    REGION Cartesian_Jog
        // HMI jog buttons -> GDB_AxisCtrl.LKinCtrl.input.jogframe Cartesian
        // direction bits. WCS frame jog: the 4 HMI axis-pairs drive
        // X (J1 buttons) / Y (J2) / Z (J3) / A (J4). XOR safety - if both
        // forward + backward are held, neither wins. Each bit is ANDed with
        // statManualOK, so leaving manual mode forces every jog bit FALSE.
        // SCARA is 4-DOF: the B / C jog directions are held FALSE.
        "GDB_AxisCtrl".LKinCtrl.input.jogframe."jogX+" := #statManualOK AND "GDB_ManualCmd".bo_J1_JogForward  AND NOT "GDB_ManualCmd".bo_J1_JogBackward;
        "GDB_AxisCtrl".LKinCtrl.input.jogframe."jogX-" := #statManualOK AND "GDB_ManualCmd".bo_J1_JogBackward AND NOT "GDB_ManualCmd".bo_J1_JogForward;
        "GDB_AxisCtrl".LKinCtrl.input.jogframe."jogY+" := #statManualOK AND "GDB_ManualCmd".bo_J2_JogForward  AND NOT "GDB_ManualCmd".bo_J2_JogBackward;
        "GDB_AxisCtrl".LKinCtrl.input.jogframe."jogY-" := #statManualOK AND "GDB_ManualCmd".bo_J2_JogBackward AND NOT "GDB_ManualCmd".bo_J2_JogForward;
        "GDB_AxisCtrl".LKinCtrl.input.jogframe."jogZ+" := #statManualOK AND "GDB_ManualCmd".bo_J3_JogForward  AND NOT "GDB_ManualCmd".bo_J3_JogBackward;
        "GDB_AxisCtrl".LKinCtrl.input.jogframe."jogZ-" := #statManualOK AND "GDB_ManualCmd".bo_J3_JogBackward AND NOT "GDB_ManualCmd".bo_J3_JogForward;
        "GDB_AxisCtrl".LKinCtrl.input.jogframe."jogA+" := #statManualOK AND "GDB_ManualCmd".bo_J4_JogForward  AND NOT "GDB_ManualCmd".bo_J4_JogBackward;
        "GDB_AxisCtrl".LKinCtrl.input.jogframe."jogA-" := #statManualOK AND "GDB_ManualCmd".bo_J4_JogBackward AND NOT "GDB_ManualCmd".bo_J4_JogForward;
        "GDB_AxisCtrl".LKinCtrl.input.jogframe."jogB+" := FALSE;
        "GDB_AxisCtrl".LKinCtrl.input.jogframe."jogB-" := FALSE;
        "GDB_AxisCtrl".LKinCtrl.input.jogframe."jogC+" := FALSE;
        "GDB_AxisCtrl".LKinCtrl.input.jogframe."jogC-" := FALSE;
    END_REGION

    REGION Kin_Manual_Move
        // bo_KinGo rising edge -> a point-to-point move to the operator-set
        // (cfgKinTargetX/Y/Z/A) via the shared movelinear interface (the
        // OB30 axis layer runs the MC). The R_TRIG runs every scan; the move
        // is issued only in manual mode. bo_execute is held until FB_AxisCtrl
        // reports the move done. Manual dynamics: 200 mm/s (auto cycle: 300).
        #sRTRIGKinGo(CLK := "GDB_ManualCmd".bo_KinGo);
        IF #statManualOK THEN
            IF #sRTRIGKinGo.Q THEN
                "GDB_AxisCtrl".LKinCtrl.input.movelinear.targetposition.x := "GDB_ManualCmd".cfgKinTargetX;
                "GDB_AxisCtrl".LKinCtrl.input.movelinear.targetposition.y := "GDB_ManualCmd".cfgKinTargetY;
                "GDB_AxisCtrl".LKinCtrl.input.movelinear.targetposition.z := "GDB_ManualCmd".cfgKinTargetZ;
                "GDB_AxisCtrl".LKinCtrl.input.movelinear.targetposition.a := "GDB_ManualCmd".cfgKinTargetA;
                "GDB_AxisCtrl".LKinCtrl.input.movelinear.targetposition.b := 0.0;
                "GDB_AxisCtrl".LKinCtrl.input.movelinear.targetposition.c := 0.0;
                "GDB_AxisCtrl".LKinCtrl.input.movelinear.r64_velocity     := 200.0;
                "GDB_AxisCtrl".LKinCtrl.input.movelinear.r64_acceleration := 2000.0;
                "GDB_AxisCtrl".LKinCtrl.input.movelinear.r64_deceleration := 2000.0;
                "GDB_AxisCtrl".LKinCtrl.input.movelinear.r64_jerk         := 20000.0;
                "GDB_AxisCtrl".LKinCtrl.input.movelinear.bo_isPTP         := FALSE;
                "GDB_AxisCtrl".LKinCtrl.input.movelinear.bo_execute       := TRUE;
            END_IF;
            // drop the execute hold once the OB30 axis layer reports done
            IF "GDB_AxisCtrl".LKinCtrl.output.movelinear.bo_done THEN
                "GDB_AxisCtrl".LKinCtrl.input.movelinear.bo_execute := FALSE;
            END_IF;
        END_IF;
    END_REGION

    REGION Status_Mirror
        // TO StatusWord bits + GDB_AxisCtrl outputs -> GDB_ManualStatus.
        // Runs every scan (NOT gated on statManualOK) so HMI lamps show the
        // truth regardless of mode. StatusWord (Siemens TO_PositioningAxis
        // MC 9.0): %X1 = Error, %X5 = Homed, %X7 = Standstill (NOT-%X7 =
        // motion in progress). Group power is all-or-nothing
        // (LKinCtrl_MC_GroupPower) - all 4 joints mirror the group bo_enabled.
        "GDB_ManualStatus".bo_J1_Enabled := "GDB_AxisCtrl".LKinCtrl.output.bo_enabled;
        "GDB_ManualStatus".bo_J2_Enabled := "GDB_AxisCtrl".LKinCtrl.output.bo_enabled;
        "GDB_ManualStatus".bo_J3_Enabled := "GDB_AxisCtrl".LKinCtrl.output.bo_enabled;
        "GDB_ManualStatus".bo_J4_Enabled := "GDB_AxisCtrl".LKinCtrl.output.bo_enabled;

        "GDB_ManualStatus".bo_J1_Homed := "J1_SCARA_Arm3D".StatusWord.%X5;
        "GDB_ManualStatus".bo_J2_Homed := "J2_SCARA_Arm3D".StatusWord.%X5;
        "GDB_ManualStatus".bo_J3_Homed := "J3_SCARA_Arm3D".StatusWord.%X5;
        "GDB_ManualStatus".bo_J4_Homed := "J4_SCARA_Arm3D".StatusWord.%X5;

        "GDB_ManualStatus".bo_J1_Error := "J1_SCARA_Arm3D".StatusWord.%X1;
        "GDB_ManualStatus".bo_J2_Error := "J2_SCARA_Arm3D".StatusWord.%X1;
        "GDB_ManualStatus".bo_J3_Error := "J3_SCARA_Arm3D".StatusWord.%X1;
        "GDB_ManualStatus".bo_J4_Error := "J4_SCARA_Arm3D".StatusWord.%X1;

        "GDB_ManualStatus".bo_J1_JogActive := NOT "J1_SCARA_Arm3D".StatusWord.%X7;
        "GDB_ManualStatus".bo_J2_JogActive := NOT "J2_SCARA_Arm3D".StatusWord.%X7;
        "GDB_ManualStatus".bo_J3_JogActive := NOT "J3_SCARA_Arm3D".StatusWord.%X7;
        "GDB_ManualStatus".bo_J4_JogActive := NOT "J4_SCARA_Arm3D".StatusWord.%X7;

        "GDB_ManualStatus".bo_KinEnabled := "GDB_AxisCtrl".LKinCtrl.output.bo_enabled;
        "GDB_ManualStatus".bo_KinHomed   := "GDB_AxisCtrl".LKinCtrl.output.bo_homed;
        "GDB_ManualStatus".bo_KinError   := "GDB_AxisCtrl".LKinCtrl.output.bo_fault;
        "GDB_ManualStatus".bo_KinReady   := "GDB_AxisCtrl".LKinCtrl.output.bo_ready;
        "GDB_ManualStatus".bo_KinManualBusy := "GDB_AxisCtrl".LKinCtrl.output.movelinear.bo_busy;
    END_REGION

END_FUNCTION_BLOCK

FUNCTION_BLOCK "FB_Init"
{ S7_Optimized_Access := 'TRUE' }
VERSION : 1.0
// =====================================================================
// SCARA ABCDE — Initialization / Homing  (Phase 3, 2026-05-21)
//
// Dedicated init/homing block per the 2026-05-21 TIA programming review
// (§1.4): homing must NOT live inside FB_AutoCtrl. Belongs to the 600
// axis/kinematics layer and runs in OB30 (10 ms cyclic interrupt),
// alongside FB_AxisCtrl.
//
// Homes the SCARA kinematics group via the library FB
// LKinCtrl_MC_GroupHome, which fires MC_HOME on every axis of ScaraArm3D
// from a per-axis mode[] + position[] array — read straight from the
// consolidated GDB_AxisCtrl.LKinCtrl.input.configuration.home struct.
//
// Two home types (review item E) — selected by the i16_mode[] value
// (the HMI / Startup OB sets it; FB_Init is mode-agnostic):
//   mode = 5  "go to zero position" — MC_Home active homing: each axis
//             runs its configured homing movement and ends at the TO
//             <TO>.Homing.HomePosition.
//   mode = 7  "set current as home" — MC_Home absolute-encoder
//             adjustment (absolute): current position set to
//             position[i], offset stored retentively. Correct for the
//             SCARA's absolute encoders (Sensor[1].Type = 2); no motion.
//
// Trigger: rising edge of GDB_AxisCtrl.LKinCtrl.input.bo_home (the HMI
// Home button). LKinCtrl_MC_GroupHome edge-detects 'execute' internally.
//
// TODO (Phase 3 refinement): for mode = 5 active homing, sequence the
// per-axis homing order + speeds (the review asks for an explicit axis
// order). LKinCtrl_MC_GroupHome homes all axes concurrently; for the
// no-motion mode = 7 case (the SCARA default) concurrent is correct.
// =====================================================================
   VAR
      instGroupHome : "LKinCtrl_MC_GroupHome";
   END_VAR


BEGIN

    REGION Group_Homing
        // Home all kinematic axes. position[]/mode[] come from the
        // consolidated GDB_AxisCtrl config; the HMI sets mode = 5 or 7
        // to choose the home type before pulsing bo_home.
        #instGroupHome(execute   := "GDB_AxisCtrl".LKinCtrl.input.bo_home,
                       position  := "GDB_AxisCtrl".LKinCtrl.input.configuration.home.r64_homeposition,
                       mode      := "GDB_AxisCtrl".LKinCtrl.input.configuration.home.i16_mode,
                       axesGroup := "ScaraArm3D");

        // Homed status: cleared while homing runs, latched TRUE on done.
        IF #instGroupHome.busy THEN
            "GDB_AxisCtrl".LKinCtrl.output.bo_homed := FALSE;
        END_IF;
        IF #instGroupHome.done THEN
            "GDB_AxisCtrl".LKinCtrl.output.bo_homed := TRUE;
        END_IF;
    END_REGION

END_FUNCTION_BLOCK

FUNCTION_BLOCK "LKinCtrl_MC_GroupHome"
TITLE = LKinCtrl_MC_GroupHome
{ S7_Optimized_Access := 'TRUE' }
AUTHOR : 'handling.team.automation@siemens.com'
FAMILY : LKinCtrl
VERSION : 5.0
//FB provides funcitonalities to home all axes (TO_PositioningAxis or TO_SynchronousAxis) interconnected with TO Kinematics
   VAR_INPUT 
      execute : Bool;   // Rising edge starts action once
      position : Array[1..#MAX_NO_OF_AXES] of LReal;   // reference positions / orientations
      mode : Array[1..#MAX_NO_OF_AXES] of Int;   // homing modes for each axis
   END_VAR

   VAR_OUTPUT 
      done { ExternalWritable := 'False'} : Bool;   // axesGroup successfully referenced
      busy { ExternalWritable := 'False'} : Bool;   // FB is not finished and new output values can be expected
      active { ExternalWritable := 'False'} : Bool;   // FB in control of axesGroup / kinematic in motion
      commandAborted { ExternalWritable := 'False'} : Bool;   // command is aborted by another command
      error { ExternalWritable := 'False'} : Bool;   // an error occurred during the execution of the FB
      diagnostics { ExternalWritable := 'False'} : "LKinCtrl_typeAuxFCDiagnostics";   // diagnostics information of FB (optional)
   END_VAR

   VAR_IN_OUT 
      axesGroup {InstructionName := 'TO_Kinematics'; LibVersion := '9.0'} : TO_Kinematics;   // reference to the axesGroup
   END_VAR

   VAR 
      statExecuteOld { ExternalAccessible := 'False'; ExternalVisible := 'False'; ExternalWritable := 'False'} : Bool;   // Old value of 'execute' input for edge detection
      statDone { ExternalAccessible := 'False'; ExternalVisible := 'False'; ExternalWritable := 'False'} : Bool;   // Static value for output 'done'
      statBusy { ExternalAccessible := 'False'; ExternalVisible := 'False'; ExternalWritable := 'False'} : Bool;   // Static value for output 'busy'
      statError { ExternalAccessible := 'False'; ExternalVisible := 'False'; ExternalWritable := 'False'} : Bool;   // Static value for output 'error'
      statCommandAborted { ExternalAccessible := 'False'; ExternalVisible := 'False'; ExternalWritable := 'False'} : Bool;   // Static value for output 'commandAborted'
      statStatus { ExternalAccessible := 'False'; ExternalVisible := 'False'; ExternalWritable := 'False'} : Word := #STATUS_NO_CALL;   // Static value for output 'status'
      statSubfunctionStatus { ExternalAccessible := 'False'; ExternalVisible := 'False'; ExternalWritable := 'False'} : Word;   // Static value for output 'subFunctionStatus'
      statAxisNumberDiag { ExternalAccessible := 'False'; ExternalVisible := 'False'; ExternalWritable := 'False'} : Int;   // Static value for output 'axisNumber'
      statErrorDetailNumber { ExternalAccessible := 'False'; ExternalVisible := 'False'; ExternalWritable := 'False'} : UDInt;   // static to store axis error detail number
      statStateMachine { ExternalAccessible := 'False'; ExternalVisible := 'False'; ExternalWritable := 'False'} : DInt := #FB_STATE_NO_PROCESSING;   // State in the state machine of the FB
      statInitInstances { ExternalAccessible := 'False'; ExternalVisible := 'False'; ExternalWritable := 'False'} : Bool;   // Static value to initialize all instances
      statExsitingAxesCtr { ExternalAccessible := 'False'; ExternalVisible := 'False'; ExternalWritable := 'False'} : Int;   // static counter for existing axes
      statHomedAxesCtr { ExternalAccessible := 'False'; ExternalVisible := 'False'; ExternalWritable := 'False'} : Int;   // static counter for successfully homed axes
      statAxes { ExternalAccessible := 'False'; ExternalVisible := 'False'; ExternalWritable := 'False'} : Array[1..#MAX_NO_OF_AXES] of DB_ANY;   // array of struct containing axis DB_ANY and type of axis
      statHomePos { ExternalAccessible := 'False'; ExternalVisible := 'False'; ExternalWritable := 'False'} : Array[1..#MAX_NO_OF_AXES] of LReal;   // reference positions / orientations
      instMCHome {InstructionName := 'MC_HOME'; LibVersion := '9.0'; ExternalAccessible := 'False'; ExternalVisible := 'False'; ExternalWritable := 'False'; S7_SetPoint := 'False'} : Array[1..#MAX_NO_OF_AXES] of MC_HOME;   // multi instance array of MC_HOME
   END_VAR

   VAR_TEMP 
      tempExecute : Bool;   // temporary value for input 'execute'
      tempAxisCtr : Int;   // temporary counter variable for axes
      tempRefToAxis {InstructionName := 'TO_PositioningAxis'; LibVersion := '9.0'} : REF_TO TO_PositioningAxis;   // temporary reference to axis
   END_VAR

   VAR CONSTANT 
      FB_STATE_NO_PROCESSING : DInt := 0;   // state machine constant
      CALC_HOME_POS : DInt := 10;   // state machine constant
      HOMING_IN_PROGRESS : DInt := 20;   // state machine constant
      MAX_NO_OF_AXES : Int := 6;   // maximum number of axes
      STATUS_EXECUTION_FINISHED : Word := 16#0000;   // Execution finished without errors
      STATUS_NO_CALL : Word := 16#7000;   // No job being currently processed
      STATUS_FIRST_CALL : Word := 16#7001;   // First call after incoming new job (rising edge 'execute')
      STATUS_SUBSEQUENT_CALL : Word := 16#7002;   // Subsequent call during active processing without further details
      STATUS_COMMAND_ABORTED : Word := 16#7FFF;   // commanded functionality has been aborted by another command
      ERR_AXIS_ERROR : Word := 16#8350;   // error pending at axis
      ERR_MC_HOME : Word := 16#8351;   // error during execution of MC_HOME for axis
      ERR_AXIS_REF : Word := 16#8373;   // error due to missing axis reference
      ERR_UNDEFINED_STATE : Word := 16#8600;   // error due to an undefined state in state machine
   END_VAR


BEGIN
	//==========================================================================================
	// SIEMENS AG
	// (c)Copyright 2019 All Rights Reserved
	//------------------------------------------------------------------------------------------
	// Library: LKinCtrl
	// Tested with: S7-1517T-3 PN/DP
	// Engineering: TIA Portal V18
	// Restrictions: ---
	// Requirements: S7-1500T FW 3.0
	// Functionality: LKinCtrl_MC_GroupHome
	// The FB is executing MC_HOME function blocks to reference all axes
	// corresponding to a specific axesGroup (TO Kinematics)
	//
	// Support: tech.team.motioncontrol@siemens.com
	// Note: Parameter comments are only available in language 'English (United States)'
	//------------------------------------------------------------------------------------------
	// Change log table:
	// Version    Date          Expert in charge    Changes applied
	// 01.00.00   26.02.2019    JR                  First release version v1.0
	// 01.01.00   13.10.2022    FR                  Reworked with REF_TO
	//===========================================================================================
	
	#tempExecute := #execute; // Work with temporary value / create process image
	
	REGION TRIGGERING
	  IF (#tempExecute = TRUE) AND (#statExecuteOld = FALSE) // Check if FB is triggered
	  THEN // First call; initialize FB
	    #statDone := FALSE;
	    #statBusy := TRUE;
	    #statError := FALSE;
	    #statStatus := #STATUS_FIRST_CALL;
	    
	    #statStateMachine := #CALC_HOME_POS; // State machine - start processing
	    
	    // Initialize functionality: reset of variables, diagnostics, etc.
	    #statErrorDetailNumber := 0;
	    #statAxisNumberDiag := 0;
	    #statSubfunctionStatus := 16#0;
	    #statInitInstances := TRUE;
	    // Reset home position
	    FOR #tempAxisCtr := 1 TO #MAX_NO_OF_AXES DO
	      #statHomePos[#tempAxisCtr] := 0;
	    END_FOR;
	    
	    // Initialize functionality: call subsidiary FBs with FALSE
	    // assign DB number of connected axis to DB_ANY type
	    #statAxes[1] := #axesGroup.KinematicsAxis.A1;
	    #statAxes[2] := #axesGroup.KinematicsAxis.A2;
	    #statAxes[3] := #axesGroup.KinematicsAxis.A3;
	    #statAxes[4] := #axesGroup.KinematicsAxis.A4;
	    #statAxes[5] := #axesGroup.KinematicsAxis.A5;
	    #statAxes[6] := #axesGroup.KinematicsAxis.A6;
	    
	  ELSIF (#statStatus = #STATUS_FIRST_CALL) THEN
	    #statStatus := #STATUS_SUBSEQUENT_CALL;
	  END_IF;
	  
	  // Edge detection 'execute' input
	  #statExecuteOld := #tempExecute;
	END_REGION TRIGGERING
	
	IF (#statStatus = #STATUS_NO_CALL) THEN
	  // Nothing to do -> End here to reduce "system load"
	  RETURN;
	END_IF;
	
	REGION STATE_MACHINE
	  CASE #statStateMachine OF // State machine of FB
	    #FB_STATE_NO_PROCESSING: // No processing active (Note: this state must always be present and left empty)
	      ;
	      
	    #CALC_HOME_POS:
	      REGION CALC_HOME_POS
	        // calculations for homing positions according to coordSystem added later
	        #statHomePos := #position;
	        
	        // go to next state
	        #statStateMachine := #HOMING_IN_PROGRESS;
	      END_REGION CALC_HOME_POS
	      
	    #HOMING_IN_PROGRESS:
	      REGION HOMING_IN_PROGRESS
	        IF #statInitInstances = FALSE THEN
	          // set to next state but overwrite if one instance of MC_Home is still busy 
	          #statStatus := #STATUS_EXECUTION_FINISHED;
	        END_IF;
	        
	        FOR #tempAxisCtr := 1 TO #MAX_NO_OF_AXES DO
	          // To init MC_Home, call with execute=FALSE in first cycle
	          #instMCHome[#tempAxisCtr].Execute := NOT #statInitInstances;
	          
	          // Check if axis is used
	          IF #statAxes[#tempAxisCtr] = 0 THEN
	            CONTINUE;
	          END_IF;
	          
	          // Cast
	          #tempRefToAxis ?= #statAxes[#tempAxisCtr];
	          
	          // Check if cast is valid
	          IF #tempRefToAxis = NULL THEN
	            // set status
	            #statStatus := #ERR_AXIS_REF;
	            // write axis number to diagnostics
	            #statAxisNumberDiag := #tempAxisCtr;
	            EXIT;
	          END_IF;
	          
	          // check for no error to be pending
	          IF #statStatus.%X15 = FALSE THEN
	            // Call mc_reset
	            #instMCHome[#tempAxisCtr](Axis     := #tempRefToAxis^,
	                                      Position := #statHomePos[#tempAxisCtr],
	                                      Mode     := #mode[#tempAxisCtr]);
	            
	            // check for homing to be busy
	            IF #instMCHome[#tempAxisCtr].Busy THEN
	              // stay in this state if busy
	              #statStatus := #STATUS_SUBSEQUENT_CALL;
	            ELSIF #instMCHome[#tempAxisCtr].Error OR #instMCHome[#tempAxisCtr].CommandAborted THEN
	              // set status
	              #statStatus := #ERR_MC_HOME;
	              // write MC_POWER errorID to diagnostics
	              #statSubfunctionStatus := #instMCHome[#tempAxisCtr].ErrorId;
	              // write axis number to diagnostics
	              #statAxisNumberDiag := #tempAxisCtr;
	              // exit loop once error is found
	              EXIT;
	            END_IF;
	          END_IF;
	        END_FOR;
	        
	        // Reset init bit
	        #statInitInstances := FALSE;
	      END_REGION HOMING_IN_PROGRESS
	      
	    ELSE // Undefined state in state machine reached
	      #statStatus := #ERR_UNDEFINED_STATE;
	  END_CASE;
	END_REGION STATE_MACHINE
	
	REGION OUTPUTS
	  // Write outputs
	  IF (#statStatus = #STATUS_EXECUTION_FINISHED) AND (#statDone = FALSE) THEN // Execution finished without errors
	    #statDone := TRUE;
	    #statBusy := FALSE;
	    #statError := FALSE;
	    #statStateMachine := #FB_STATE_NO_PROCESSING; // Switch state machine to "no processing"
	    
	  ELSIF (#statStatus.%X15 = TRUE) AND (#statError = FALSE) THEN // Error occurred (#statStatus is 16#8000 to 16#FFFF)
	    #statDone := FALSE;
	    #statBusy := FALSE;
	    #statError := TRUE;
	    #statStateMachine := #FB_STATE_NO_PROCESSING; // Switch state machine to "no processing"
	    
	  ELSIF (#tempExecute = FALSE) AND ((#statDone = TRUE) OR (#statError = TRUE)) THEN // Reset outputs
	    #statDone := FALSE;
	    #statBusy := FALSE;
	    #statError := FALSE;
	    #statStatus := #STATUS_NO_CALL;
	  END_IF;
	  
	  // Write static values to outputs
	  #done := #statDone;
	  #busy := #statBusy;
	  #error := #statError;
	  #diagnostics.status := #statStatus;
	  #diagnostics.subfunctionStatus := #statSubfunctionStatus;
	  #diagnostics.axisNumber := #statAxisNumberDiag;
	  #diagnostics.errorDetail := #statErrorDetailNumber;
	  #diagnostics.stateNumber := #statStateMachine;
	END_REGION OUTPUTS
	
	// =================================================================================================================
	// End of Function Block: LKinCtrl_MC_GroupHome
	// =================================================================================================================
END_FUNCTION_BLOCK

FUNCTION_BLOCK "FB_MovePath"
{ S7_Optimized_Access := 'TRUE' }
VERSION : 0.1

BEGIN
END_FUNCTION_BLOCK

FUNCTION_BLOCK "FB_PatternAutoGen"
{ S7_Optimized_Access := 'TRUE' }
VERSION : 3.0
// =====================================================================
// SCARA Phase 2 Modules D + E - one-block auto-pattern generator with
// dual-pallet selection.  (V3.0, 2026-05-23 - WanErXin review fixes)
//
// MODULE D (V1.0, 2026-05-23): single-recipe one-block auto-fit. Each
// scan, validates GDB_ActiveRecipe.recipe, derives a uniform-grid pattern
// (cols/rows from pallet base + product dims), and writes the result into
// GDB_PalletizingCmd's Module-C config members for FB_AutoCtrl_Palletizing
// to consume on the next bo_InitPallet rising edge.
//
// MODULE E (V2.0, 2026-05-23): dual-pallet. recipe -> recipe1 + recipe2.
// Pallet selection is OPERATOR-DRIVEN (WanErXin pattern, no auto-advance):
// two maintained Bool flags bo_ExecutePallet1 / bo_ExecutePallet2 select
// which pallet is active. Per-pallet bo_PalletNFull alarms latch when the
// cycle completes; the just-emptied pallet's full bit auto-clears when the
// operator switches to the other side (WanErXin level-driven clear).
// FB_AutoCtrl_Palletizing remains untouched.
//
// V3.0 (2026-05-23) - critical review of WanErXin pattern surfaced 3 bugs;
// V3.0 fixes them while keeping V2.0's clean shape:
//
//   Bug #1: V2.0's LatchPalletFull used the CURRENT i16_ActivePalletIdx to
//           attribute bo_PalletDone. If the operator swapped pallets mid-
//           cycle (or released both flags), the wrong pallet's full bit
//           would latch (or neither would). FIX: snapshot activeIdx into
//           statCyclePalletIdx on the rising edge of bo_InitPallet (= the
//           moment FB_AutoCtrl_Palletizing locks aCmd[] from the current
//           GDB_PalletizingCmd config) and use that snapshot for the latch.
//
//   Bug #2: V2.0 only cleared bo_PalletNFull via the WanErXin "swap to
//           clear" path -- operator MUST go via the other pallet's button
//           to reset, even if they just physically emptied this pallet and
//           want to continue. FIX: add explicit bo_AckPallet1Full /
//           bo_AckPallet2Full HMI-write bits; while TRUE, the corresponding
//           full bit clears each scan. The WanErXin path stays as the
//           convenience alternative.
//
//   Bug #3: No aggregate "both pallets full" status for HMI / future
//           Module F-G integration. FIX: FB now computes bo_BothPalletsFull
//           = bo_Pallet1Full AND bo_Pallet2Full each scan.
//
// Each scan, in order:
//   1. ValidatePallet1: validate recipe1, compute grid, publish status echoes.
//   2. ValidatePallet2: same for recipe2.
//   3. SelectActivePallet: mutex (WanErXin) + level-driven swap-clear (WanErXin)
//      + V3.0 explicit Ack-reset (mine).
//   4. WriteActiveConfig: if active pallet 1/2 with valid recipe, write its
//      pitch/grid/dynamics into GDB_PalletizingCmd. Otherwise GDB_PalletizingCmd
//      keeps its previous state.
//   5. TrackCycleStart (V3.0): on rising edge of GDB_PalletizingCmd.bo_InitPallet,
//      snapshot tempActiveIdx into statCyclePalletIdx.
//   6. LatchPalletFull (V3.0 changed): on GDB_PalletizingCmd.bo_PalletDone,
//      latch the IN-FLIGHT pallet's full bit (via statCyclePalletIdx, not
//      current operator-driven activeIdx).
//   7. ComputeAggregate (V3.0): bo_BothPalletsFull := AND of full bits.
//
// Path ceiling: 22 boxes per pallet. Derived from GDB_PalletizingPath.aCmd[1..200]
// and the Module-C builder's (boxes * 9 + 1) commands per pallet:
// boxes_max = (200 - 1) DIV 9 = 22. Each pallet validated against the same
// ceiling (each cycle builds ONE pallet at a time).
// =====================================================================
   VAR
      // -- V3.0 cycle-attribution snapshot --
      statCyclePalletIdx  : Int;    // which pallet's cycle is in flight
      statInitPallet_prev : Bool;   // for rising-edge detection on bo_InitPallet
   END_VAR

   VAR_TEMP
      // -- pallet 1 validation + computation --
      tempPitchX1 : LReal;
      tempPitchY1 : LReal;
      tempCols1   : Int;
      tempRows1   : Int;
      tempBoxes1  : Int;
      tempValid1  : Bool;
      // -- pallet 2 validation + computation --
      tempPitchX2 : LReal;
      tempPitchY2 : LReal;
      tempCols2   : Int;
      tempRows2   : Int;
      tempBoxes2  : Int;
      tempValid2  : Bool;
      // -- pallet selection --
      tempActiveIdx : Int;
   END_VAR


BEGIN

    REGION ValidatePallet1
        #tempValid1 := "GDB_ActiveRecipe".recipe1.bo_Valid
                   AND "GDB_ActiveRecipe".recipe1.product.lr_Length     > 0.0
                   AND "GDB_ActiveRecipe".recipe1.product.lr_Width      > 0.0
                   AND "GDB_ActiveRecipe".recipe1.product.lr_Height     > 0.0
                   AND "GDB_ActiveRecipe".recipe1.product.lr_Gap        >= 0.0
                   AND "GDB_ActiveRecipe".recipe1.pallet.lr_BaseLength  > 0.0
                   AND "GDB_ActiveRecipe".recipe1.pallet.lr_BaseWidth   > 0.0
                   AND "GDB_ActiveRecipe".recipe1.pallet.i16_LayerCount >= 1
                   AND "GDB_ActiveRecipe".recipe1.dynamics.lr_Velocity     > 0.0
                   AND "GDB_ActiveRecipe".recipe1.dynamics.lr_Acceleration > 0.0
                   AND "GDB_ActiveRecipe".recipe1.dynamics.lr_Deceleration > 0.0
                   AND "GDB_ActiveRecipe".recipe1.dynamics.lr_Jerk         > 0.0;
        #tempPitchX1 := 0.0;  #tempPitchY1 := 0.0;
        #tempCols1 := 0;  #tempRows1 := 0;  #tempBoxes1 := 0;

        IF #tempValid1 THEN
            #tempPitchX1 := "GDB_ActiveRecipe".recipe1.product.lr_Length
                          + "GDB_ActiveRecipe".recipe1.product.lr_Gap;
            #tempPitchY1 := "GDB_ActiveRecipe".recipe1.product.lr_Width
                          + "GDB_ActiveRecipe".recipe1.product.lr_Gap;
            IF #tempPitchX1 > "GDB_ActiveRecipe".recipe1.pallet.lr_BaseLength
                OR #tempPitchY1 > "GDB_ActiveRecipe".recipe1.pallet.lr_BaseWidth THEN
                #tempValid1 := FALSE;
            ELSE
                #tempCols1 := LREAL_TO_INT(
                    ("GDB_ActiveRecipe".recipe1.pallet.lr_BaseLength
                     + "GDB_ActiveRecipe".recipe1.product.lr_Gap) / #tempPitchX1);
                #tempRows1 := LREAL_TO_INT(
                    ("GDB_ActiveRecipe".recipe1.pallet.lr_BaseWidth
                     + "GDB_ActiveRecipe".recipe1.product.lr_Gap) / #tempPitchY1);
                #tempBoxes1 := #tempCols1 * #tempRows1
                             * "GDB_ActiveRecipe".recipe1.pallet.i16_LayerCount;
                IF #tempCols1 < 1 OR #tempRows1 < 1 OR #tempBoxes1 > 22 THEN
                    #tempValid1 := FALSE;
                END_IF;
            END_IF;
        END_IF;

        "GDB_ActiveRecipe".bo_PatternValid1       := #tempValid1;
        "GDB_ActiveRecipe".bo_PatternError1       := NOT #tempValid1;
        "GDB_ActiveRecipe".i16_ComputedGridColsX1 := #tempCols1;
        "GDB_ActiveRecipe".i16_ComputedGridRowsY1 := #tempRows1;
        "GDB_ActiveRecipe".i16_ComputedBoxCount1  := #tempBoxes1;
    END_REGION

    REGION ValidatePallet2
        #tempValid2 := "GDB_ActiveRecipe".recipe2.bo_Valid
                   AND "GDB_ActiveRecipe".recipe2.product.lr_Length     > 0.0
                   AND "GDB_ActiveRecipe".recipe2.product.lr_Width      > 0.0
                   AND "GDB_ActiveRecipe".recipe2.product.lr_Height     > 0.0
                   AND "GDB_ActiveRecipe".recipe2.product.lr_Gap        >= 0.0
                   AND "GDB_ActiveRecipe".recipe2.pallet.lr_BaseLength  > 0.0
                   AND "GDB_ActiveRecipe".recipe2.pallet.lr_BaseWidth   > 0.0
                   AND "GDB_ActiveRecipe".recipe2.pallet.i16_LayerCount >= 1
                   AND "GDB_ActiveRecipe".recipe2.dynamics.lr_Velocity     > 0.0
                   AND "GDB_ActiveRecipe".recipe2.dynamics.lr_Acceleration > 0.0
                   AND "GDB_ActiveRecipe".recipe2.dynamics.lr_Deceleration > 0.0
                   AND "GDB_ActiveRecipe".recipe2.dynamics.lr_Jerk         > 0.0;
        #tempPitchX2 := 0.0;  #tempPitchY2 := 0.0;
        #tempCols2 := 0;  #tempRows2 := 0;  #tempBoxes2 := 0;

        IF #tempValid2 THEN
            #tempPitchX2 := "GDB_ActiveRecipe".recipe2.product.lr_Length
                          + "GDB_ActiveRecipe".recipe2.product.lr_Gap;
            #tempPitchY2 := "GDB_ActiveRecipe".recipe2.product.lr_Width
                          + "GDB_ActiveRecipe".recipe2.product.lr_Gap;
            IF #tempPitchX2 > "GDB_ActiveRecipe".recipe2.pallet.lr_BaseLength
                OR #tempPitchY2 > "GDB_ActiveRecipe".recipe2.pallet.lr_BaseWidth THEN
                #tempValid2 := FALSE;
            ELSE
                #tempCols2 := LREAL_TO_INT(
                    ("GDB_ActiveRecipe".recipe2.pallet.lr_BaseLength
                     + "GDB_ActiveRecipe".recipe2.product.lr_Gap) / #tempPitchX2);
                #tempRows2 := LREAL_TO_INT(
                    ("GDB_ActiveRecipe".recipe2.pallet.lr_BaseWidth
                     + "GDB_ActiveRecipe".recipe2.product.lr_Gap) / #tempPitchY2);
                #tempBoxes2 := #tempCols2 * #tempRows2
                             * "GDB_ActiveRecipe".recipe2.pallet.i16_LayerCount;
                IF #tempCols2 < 1 OR #tempRows2 < 1 OR #tempBoxes2 > 22 THEN
                    #tempValid2 := FALSE;
                END_IF;
            END_IF;
        END_IF;

        "GDB_ActiveRecipe".bo_PatternValid2       := #tempValid2;
        "GDB_ActiveRecipe".bo_PatternError2       := NOT #tempValid2;
        "GDB_ActiveRecipe".i16_ComputedGridColsX2 := #tempCols2;
        "GDB_ActiveRecipe".i16_ComputedGridRowsY2 := #tempRows2;
        "GDB_ActiveRecipe".i16_ComputedBoxCount2  := #tempBoxes2;
    END_REGION

    REGION SelectActivePallet
        // WanErXin mutex: one button held + other not + this side not full.
        // Both buttons / neither button / active-side full -> idle (idx 0).
        IF "GDB_ActiveRecipe".bo_ExecutePallet1
                AND NOT "GDB_ActiveRecipe".bo_ExecutePallet2
                AND NOT "GDB_ActiveRecipe".bo_Pallet1Full THEN
            #tempActiveIdx := 1;
        ELSIF "GDB_ActiveRecipe".bo_ExecutePallet2
                AND NOT "GDB_ActiveRecipe".bo_ExecutePallet1
                AND NOT "GDB_ActiveRecipe".bo_Pallet2Full THEN
            #tempActiveIdx := 2;
        ELSE
            #tempActiveIdx := 0;
        END_IF;

        "GDB_ActiveRecipe".i16_ActivePalletIdx := #tempActiveIdx;

        // WanErXin level-driven full-bit clear on operator swap:
        // operator pressing the OPPOSITE side's button (while THIS side is
        // full and THIS side's button is released) is the "I have emptied
        // this pallet, ready to re-use" gesture. Guard `AND NOT thisSide`
        // prevents a both-pressed transient from clearing prematurely.
        IF "GDB_ActiveRecipe".bo_Pallet1Full
                AND "GDB_ActiveRecipe".bo_ExecutePallet2
                AND NOT "GDB_ActiveRecipe".bo_ExecutePallet1 THEN
            "GDB_ActiveRecipe".bo_Pallet1Full := FALSE;
        END_IF;
        IF "GDB_ActiveRecipe".bo_Pallet2Full
                AND "GDB_ActiveRecipe".bo_ExecutePallet1
                AND NOT "GDB_ActiveRecipe".bo_ExecutePallet2 THEN
            "GDB_ActiveRecipe".bo_Pallet2Full := FALSE;
        END_IF;

        // V3.0 explicit Ack-reset path: operator HMI button forces this
        // side's full bit FALSE while held. Independent of the swap-clear
        // path above, so operator can reset without going via the other
        // pallet (e.g. after physically emptying and replacing the same
        // pallet station).
        IF "GDB_ActiveRecipe".bo_AckPallet1Full THEN
            "GDB_ActiveRecipe".bo_Pallet1Full := FALSE;
        END_IF;
        IF "GDB_ActiveRecipe".bo_AckPallet2Full THEN
            "GDB_ActiveRecipe".bo_Pallet2Full := FALSE;
        END_IF;
    END_REGION

    REGION WriteActiveConfig
        // Write GDB_PalletizingCmd from the active pallet's validated recipe.
        // If active is 0 (idle) OR active pallet's recipe failed validation:
        // skip the write -- GDB_PalletizingCmd keeps its previous state.
        IF #tempActiveIdx = 1 AND #tempValid1 THEN
            "GDB_PalletizingCmd".lr_BoxPitchX    := #tempPitchX1;
            "GDB_PalletizingCmd".lr_BoxPitchY    := #tempPitchY1;
            "GDB_PalletizingCmd".lr_BoxHeight    := "GDB_ActiveRecipe".recipe1.product.lr_Height;
            "GDB_PalletizingCmd".i16_GridColsX   := #tempCols1;
            "GDB_PalletizingCmd".i16_GridRowsY   := #tempRows1;
            "GDB_PalletizingCmd".i16_LayerCount  := "GDB_ActiveRecipe".recipe1.pallet.i16_LayerCount;
            "GDB_PalletizingCmd".lr_MoveVelocity := "GDB_ActiveRecipe".recipe1.dynamics.lr_Velocity;
            "GDB_PalletizingCmd".lr_MoveAccel    := "GDB_ActiveRecipe".recipe1.dynamics.lr_Acceleration;
            "GDB_PalletizingCmd".lr_MoveDecel    := "GDB_ActiveRecipe".recipe1.dynamics.lr_Deceleration;
            "GDB_PalletizingCmd".lr_MoveJerk     := "GDB_ActiveRecipe".recipe1.dynamics.lr_Jerk;
        ELSIF #tempActiveIdx = 2 AND #tempValid2 THEN
            "GDB_PalletizingCmd".lr_BoxPitchX    := #tempPitchX2;
            "GDB_PalletizingCmd".lr_BoxPitchY    := #tempPitchY2;
            "GDB_PalletizingCmd".lr_BoxHeight    := "GDB_ActiveRecipe".recipe2.product.lr_Height;
            "GDB_PalletizingCmd".i16_GridColsX   := #tempCols2;
            "GDB_PalletizingCmd".i16_GridRowsY   := #tempRows2;
            "GDB_PalletizingCmd".i16_LayerCount  := "GDB_ActiveRecipe".recipe2.pallet.i16_LayerCount;
            "GDB_PalletizingCmd".lr_MoveVelocity := "GDB_ActiveRecipe".recipe2.dynamics.lr_Velocity;
            "GDB_PalletizingCmd".lr_MoveAccel    := "GDB_ActiveRecipe".recipe2.dynamics.lr_Acceleration;
            "GDB_PalletizingCmd".lr_MoveDecel    := "GDB_ActiveRecipe".recipe2.dynamics.lr_Deceleration;
            "GDB_PalletizingCmd".lr_MoveJerk     := "GDB_ActiveRecipe".recipe2.dynamics.lr_Jerk;
        END_IF;
    END_REGION

    REGION TrackCycleStart
        // V3.0: snapshot which pallet's cycle is about to start. The Module-C
        // builder locks aCmd[] from GDB_PalletizingCmd on the rising edge of
        // bo_InitPallet, so that's the canonical "cycle started for pallet X"
        // moment. Using this snapshot (instead of the live activeIdx) means
        // mid-cycle operator swaps or releases don't mis-attribute the
        // pallet-done event in LatchPalletFull below.
        IF "GDB_PalletizingCmd".bo_InitPallet AND NOT #statInitPallet_prev THEN
            #statCyclePalletIdx := #tempActiveIdx;
        END_IF;
        #statInitPallet_prev := "GDB_PalletizingCmd".bo_InitPallet;
    END_REGION

    REGION LatchPalletFull
        // V3.0: latch the IN-FLIGHT pallet's full bit (statCyclePalletIdx),
        // not the current operator-driven activeIdx (which can change mid-
        // cycle if operator swaps or releases buttons). If statCyclePalletIdx
        // is 0 (no cycle ever started, or post-MRES), don't latch anything
        // -- the bo_PalletDone is orphan and ignored.
        IF "GDB_PalletizingCmd".bo_PalletDone THEN
            IF #statCyclePalletIdx = 1 THEN
                "GDB_ActiveRecipe".bo_Pallet1Full := TRUE;
            ELSIF #statCyclePalletIdx = 2 THEN
                "GDB_ActiveRecipe".bo_Pallet2Full := TRUE;
            END_IF;
        END_IF;
    END_REGION

    REGION ComputeAggregate
        // V3.0: single status bit for HMI / Module F-G integration to gate
        // "both pallets need unloading, robot should idle".
        "GDB_ActiveRecipe".bo_BothPalletsFull :=
            "GDB_ActiveRecipe".bo_Pallet1Full
            AND "GDB_ActiveRecipe".bo_Pallet2Full;
    END_REGION

END_FUNCTION_BLOCK

FUNCTION_BLOCK "FB_TeachCtrl"
{ S7_Optimized_Access := 'TRUE' }
VERSION : 1.2
// =====================================================================
// SCARA Phase 2 Module F - Teach mode orchestration FB  (V1.2, 2026-05-23)
//
// V1.2 fix (same-day, smoke-surfaced bug): REGION Cartesian_Jog now gates
// its 8 jogframe writes inside IF #statTeachOK THEN ... END_IF. V1.0/V1.1
// wrote them every scan as `statTeachOK AND ...`, so when teach mode was
// OFF (statTeachOK=FALSE) the writes resolved to FALSE -- and since
// FB_TeachCtrl runs AFTER FB_ManualCtrl in OB1's Auto_Cycle, those FALSE
// writes overwrote FB_ManualCtrl's TRUE jog bits, silently breaking the
// operator's manual jog whenever Module F was deployed. V1.2 keeps the
// writes when teach owns jog and leaves the register alone otherwise.
// Symmetric fix for FB_ManualCtrl is recommended but not made here
// (FB_ManualCtrl runs first; with V1.2 in place, the cross-mode jog
// interference disappears regardless).
//
// V1.1 extension (same-day): Capture path now records BOTH Cartesian TCP
// AND joint angles per Phase 2 spec §7.1 ("捕获脉冲 → 当前 TCP/关节 写点表").
// Joint angles land in GDB_TeachPoints.aJointAngles[idx, 1..4] from
// "ScaraArm3D".AxesData.A[1..4].Position (same scan as TCP capture).
// Clear / ClearAll also wipe the joint arrays. Replay currently still
// walks aPoints via Cartesian linear moves (V1.0 behavior preserved);
// joint-space PTP replay using aJointAngles is reserved for a future
// extension (per-slot bo_IsPTP flag would route here).
//
// V1.0 (2026-05-23):
// Operator-driven teach: jog the robot, capture TCP into slots, replay
// the captured sequence. Lives as the 4th mutex mode alongside ABCDE
// (GDB_MachineCmd, transitional), Palletizing (GDB_PalletizingCmd), and
// Manual (GDB_ManualCmd).
//
// REGIONs (each ~1 screen of SCL):
//   1. Mode_Gate          - statTeachOK = bo_Mode AND bo_ESTOP_LOCK AND
//                           NOT other_modes. When FALSE: idle the FSM,
//                           clear bo_execute, blank i16_TeachStep + idx.
//   2. Cartesian_Jog      - copy of FB_ManualCtrl jog wiring, gated on
//                           statTeachOK. Operator jogs in teach mode the
//                           same way as in manual mode.
//   3. Operator_Actions   - edge-detect bo_Capture / bo_Verify / bo_Clear
//                           / bo_ClearAll. Each fires once on rising edge.
//                           Capture reads actualposition (populated by
//                           FB_AxisCtrl MirrorTCP) and writes the slot.
//                           Verify pulses movelinear to drive the robot
//                           to the slot. Clear blanks the slot + flag.
//   4. Replay_FSM         - state machine triggered by bo_StartReplay.
//                           Iterates aPoints[1..16] skipping uncaptured
//                           slots; drives each via shared movelinear.
//                           Once-through; latches bo_ReplayDone at end.
//                           bo_StopReplay from any state -> idle.
//   5. Compute_PointCount - each scan, count TRUE bits in abCaptured[].
//
// The verified Module C / D / E code is untouched. FB_TeachCtrl writes
// to the shared GDB_AxisCtrl.LKinCtrl.input.{jogframe, movelinear}
// interface - same as FB_ManualCtrl and the two auto FBs - so no new MC
// instance is needed; FB_AxisCtrl (OB30) runs the actual motion.
//
// Module F 750_Teach\ namespace: GDB_TeachPoints (slot storage),
// GDB_TeachCmd (HMI commands + FB status), FB_TeachCtrl, instFB_TeachCtrl.
// =====================================================================
   VAR
      // -- operator-action edge triggers --
      sRTRIG_Capture     {InstructionName := 'R_TRIG'; LibVersion := '1.0'} : R_TRIG;
      sRTRIG_Verify      {InstructionName := 'R_TRIG'; LibVersion := '1.0'} : R_TRIG;
      sRTRIG_Clear       {InstructionName := 'R_TRIG'; LibVersion := '1.0'} : R_TRIG;
      sRTRIG_ClearAll    {InstructionName := 'R_TRIG'; LibVersion := '1.0'} : R_TRIG;
      // -- replay edge triggers --
      sRTRIG_StartReplay {InstructionName := 'R_TRIG'; LibVersion := '1.0'} : R_TRIG;
      sRTRIG_StopReplay  {InstructionName := 'R_TRIG'; LibVersion := '1.0'} : R_TRIG;
      // -- move-done edge (so each replay step advances exactly once) --
      sRTRIG_MoveDone    {InstructionName := 'R_TRIG'; LibVersion := '1.0'} : R_TRIG;
      // -- gate --
      statTeachOK : Bool;
   END_VAR

   VAR_TEMP
      tempIdxInRange : Bool;   // 1 <= i16_SlotIdx <= 16
      tempReplayIdx  : Int;    // local copy of i16_ReplayIdx for FSM scratch
      tempCount      : Int;    // for the PointCount loop
      i              : Int;    // generic loop counter
   END_VAR


BEGIN

    REGION Mode_Gate
        // 4-way mutex. Teach is the 4th mode. GDB_MachineCmd.bo_Mode is
        // transitional (ABCDE demo, slated for deletion); the term decays
        // to a no-op once ABCDE is removed.
        #statTeachOK := "GDB_TeachCmd".bo_Mode
                        AND "GDB_TeachCmd".bo_ESTOP_LOCK
                        AND NOT "GDB_MachineCmd".bo_Mode
                        AND NOT "GDB_PalletizingCmd".bo_Mode
                        AND NOT "GDB_ManualCmd".bo_Mode;

        // On mode exit: clean idle. Clear FSM state and any held execute.
        IF NOT #statTeachOK THEN
            IF "GDB_TeachCmd".i16_TeachStep <> 0 THEN
                "GDB_TeachCmd".i16_TeachStep := 0;
                "GDB_TeachCmd".i16_ReplayIdx := 0;
                "GDB_AxisCtrl".LKinCtrl.input.movelinear.bo_execute := FALSE;
            END_IF;
        END_IF;

        // Edge detectors always run (R_TRIG must see edges in real-time
        // to not miss them); the action gates below check #statTeachOK.
        #sRTRIG_Capture(    CLK := "GDB_TeachCmd".bo_Capture);
        #sRTRIG_Verify(     CLK := "GDB_TeachCmd".bo_Verify);
        #sRTRIG_Clear(      CLK := "GDB_TeachCmd".bo_Clear);
        #sRTRIG_ClearAll(   CLK := "GDB_TeachCmd".bo_ClearAll);
        #sRTRIG_StartReplay(CLK := "GDB_TeachCmd".bo_StartReplay);
        #sRTRIG_StopReplay( CLK := "GDB_TeachCmd".bo_StopReplay);
        #sRTRIG_MoveDone(   CLK := "GDB_AxisCtrl".LKinCtrl.output.movelinear.bo_done);

        // Range-check the slot index (nested IF, per SCL-no-short-circuit
        // rule for array access). Used by Capture/Verify/Clear below.
        #tempIdxInRange := FALSE;
        IF "GDB_TeachCmd".i16_SlotIdx >= 1 THEN
            IF "GDB_TeachCmd".i16_SlotIdx <= 16 THEN
                #tempIdxInRange := TRUE;
            END_IF;
        END_IF;
    END_REGION

    REGION Cartesian_Jog
        // Mirror of FB_ManualCtrl REGION Cartesian_Jog: the same HMI jog
        // buttons (bo_J1_JogForward .. bo_J4_JogBackward) drive Cartesian
        // X/Y/Z/A. XOR safety: both directions held -> neither wins.
        // SCARA is 4-DOF, so B/C jog held FALSE.
        //
        // V1.2 (smoke-surfaced fix): the writes are GATED by IF #statTeachOK
        // because FB_TeachCtrl runs AFTER FB_ManualCtrl in OB1 (Manual_Control
        // before Auto_Cycle/Teach_Cycle). V1.0/V1.1 wrote `#statTeachOK AND ...`
        // every scan -- when teach was OFF, that resolved to FALSE and
        // overwrote any TRUE bits FB_ManualCtrl had set, silently breaking
        // the operator's manual jog. With the IF-gate, FB_TeachCtrl simply
        // doesn't touch jogframe when teach is off, leaving FB_ManualCtrl's
        // writes as the authoritative value. When teach IS active, manual
        // mode is mutex-blocked (statManualOK FALSE -> FB_ManualCtrl writes
        // all FALSE), so FB_TeachCtrl's writes win uncontested.
        IF #statTeachOK THEN
            "GDB_AxisCtrl".LKinCtrl.input.jogframe."jogX+" := "GDB_ManualCmd".bo_J1_JogForward  AND NOT "GDB_ManualCmd".bo_J1_JogBackward;
            "GDB_AxisCtrl".LKinCtrl.input.jogframe."jogX-" := "GDB_ManualCmd".bo_J1_JogBackward AND NOT "GDB_ManualCmd".bo_J1_JogForward;
            "GDB_AxisCtrl".LKinCtrl.input.jogframe."jogY+" := "GDB_ManualCmd".bo_J2_JogForward  AND NOT "GDB_ManualCmd".bo_J2_JogBackward;
            "GDB_AxisCtrl".LKinCtrl.input.jogframe."jogY-" := "GDB_ManualCmd".bo_J2_JogBackward AND NOT "GDB_ManualCmd".bo_J2_JogForward;
            "GDB_AxisCtrl".LKinCtrl.input.jogframe."jogZ+" := "GDB_ManualCmd".bo_J3_JogForward  AND NOT "GDB_ManualCmd".bo_J3_JogBackward;
            "GDB_AxisCtrl".LKinCtrl.input.jogframe."jogZ-" := "GDB_ManualCmd".bo_J3_JogBackward AND NOT "GDB_ManualCmd".bo_J3_JogForward;
            "GDB_AxisCtrl".LKinCtrl.input.jogframe."jogA+" := "GDB_ManualCmd".bo_J4_JogForward  AND NOT "GDB_ManualCmd".bo_J4_JogBackward;
            "GDB_AxisCtrl".LKinCtrl.input.jogframe."jogA-" := "GDB_ManualCmd".bo_J4_JogBackward AND NOT "GDB_ManualCmd".bo_J4_JogForward;
            "GDB_AxisCtrl".LKinCtrl.input.jogframe."jogB+" := FALSE;
            "GDB_AxisCtrl".LKinCtrl.input.jogframe."jogB-" := FALSE;
            "GDB_AxisCtrl".LKinCtrl.input.jogframe."jogC+" := FALSE;
            "GDB_AxisCtrl".LKinCtrl.input.jogframe."jogC-" := FALSE;
        END_IF;
        // When NOT #statTeachOK: no writes -- leave jogframe alone so
        // FB_ManualCtrl (or whoever else, future) owns it.
    END_REGION

    REGION Operator_Actions
        // --- Capture (V1.1): snapshot BOTH live TCP AND joint angles ---
        IF #sRTRIG_Capture.Q AND #statTeachOK AND #tempIdxInRange THEN
            // (a) Cartesian TCP -> aPoints[idx]. LKinCtrl_typePoint.position is
            //     [0..5] but SCARA is 4-DOF -- b/c populated from TO too (the
            //     kinematics solver fills them based on joint posture).
            "GDB_TeachPoints".aPoints["GDB_TeachCmd".i16_SlotIdx].position[0] := "GDB_AxisCtrl".LKinCtrl.output.actualposition.x;
            "GDB_TeachPoints".aPoints["GDB_TeachCmd".i16_SlotIdx].position[1] := "GDB_AxisCtrl".LKinCtrl.output.actualposition.y;
            "GDB_TeachPoints".aPoints["GDB_TeachCmd".i16_SlotIdx].position[2] := "GDB_AxisCtrl".LKinCtrl.output.actualposition.z;
            "GDB_TeachPoints".aPoints["GDB_TeachCmd".i16_SlotIdx].position[3] := "GDB_AxisCtrl".LKinCtrl.output.actualposition.a;
            "GDB_TeachPoints".aPoints["GDB_TeachCmd".i16_SlotIdx].position[4] := "GDB_AxisCtrl".LKinCtrl.output.actualposition.b;
            "GDB_TeachPoints".aPoints["GDB_TeachCmd".i16_SlotIdx].position[5] := "GDB_AxisCtrl".LKinCtrl.output.actualposition.c;
            "GDB_TeachPoints".aPoints["GDB_TeachCmd".i16_SlotIdx].coordSystem := 0;  // WCS
            // (b) Joint angles J1..J4 -> aJointAngles[idx, joint] (V1.1, Phase 2 §7.1).
            //     Same source FB_MCDDataTransfer uses for the kin-group-view mirror.
            //     2D array: comma-indexed (S7-1500T doesn't allow nested Array-of-
            //     Array in interface declarations).
            "GDB_TeachPoints".aJointAngles["GDB_TeachCmd".i16_SlotIdx, 1] := "ScaraArm3D".AxesData.A[1].Position;
            "GDB_TeachPoints".aJointAngles["GDB_TeachCmd".i16_SlotIdx, 2] := "ScaraArm3D".AxesData.A[2].Position;
            "GDB_TeachPoints".aJointAngles["GDB_TeachCmd".i16_SlotIdx, 3] := "ScaraArm3D".AxesData.A[3].Position;
            "GDB_TeachPoints".aJointAngles["GDB_TeachCmd".i16_SlotIdx, 4] := "ScaraArm3D".AxesData.A[4].Position;
            "GDB_TeachPoints".abCaptured["GDB_TeachCmd".i16_SlotIdx] := TRUE;
            "GDB_TeachCmd".i16_TeachStep := 10;  // HMI feedback (one scan)
        ELSIF "GDB_TeachCmd".i16_TeachStep = 10 THEN
            "GDB_TeachCmd".i16_TeachStep := 0;  // auto-clear after capture flash
        END_IF;

        // --- Verify: move robot to aPoints[SlotIdx] ---
        IF #sRTRIG_Verify.Q AND #statTeachOK AND #tempIdxInRange THEN
            IF "GDB_TeachPoints".abCaptured["GDB_TeachCmd".i16_SlotIdx] THEN
                "GDB_AxisCtrl".LKinCtrl.input.movelinear.targetposition.x := "GDB_TeachPoints".aPoints["GDB_TeachCmd".i16_SlotIdx].position[0];
                "GDB_AxisCtrl".LKinCtrl.input.movelinear.targetposition.y := "GDB_TeachPoints".aPoints["GDB_TeachCmd".i16_SlotIdx].position[1];
                "GDB_AxisCtrl".LKinCtrl.input.movelinear.targetposition.z := "GDB_TeachPoints".aPoints["GDB_TeachCmd".i16_SlotIdx].position[2];
                "GDB_AxisCtrl".LKinCtrl.input.movelinear.targetposition.a := "GDB_TeachPoints".aPoints["GDB_TeachCmd".i16_SlotIdx].position[3];
                "GDB_AxisCtrl".LKinCtrl.input.movelinear.targetposition.b := 0.0;
                "GDB_AxisCtrl".LKinCtrl.input.movelinear.targetposition.c := 0.0;
                "GDB_AxisCtrl".LKinCtrl.input.movelinear.r64_velocity     := "GDB_TeachCmd".lr_ReplayVel;
                "GDB_AxisCtrl".LKinCtrl.input.movelinear.r64_acceleration := 2000.0;
                "GDB_AxisCtrl".LKinCtrl.input.movelinear.r64_deceleration := 2000.0;
                "GDB_AxisCtrl".LKinCtrl.input.movelinear.r64_jerk         := 20000.0;
                "GDB_AxisCtrl".LKinCtrl.input.movelinear.bo_isPTP         := FALSE;
                "GDB_AxisCtrl".LKinCtrl.input.movelinear.bo_execute       := TRUE;
                "GDB_TeachCmd".i16_TeachStep := 20;  // verify-in-flight
            END_IF;
        END_IF;
        // Verify drop: when move reports done, drop execute and return to idle.
        IF "GDB_TeachCmd".i16_TeachStep = 20 AND #sRTRIG_MoveDone.Q THEN
            "GDB_AxisCtrl".LKinCtrl.input.movelinear.bo_execute := FALSE;
            "GDB_TeachCmd".i16_TeachStep := 0;
        END_IF;

        // --- Clear single slot (V1.1: zero BOTH TCP and joint arrays) ---
        IF #sRTRIG_Clear.Q AND #statTeachOK AND #tempIdxInRange THEN
            "GDB_TeachPoints".aPoints["GDB_TeachCmd".i16_SlotIdx].position[0] := 0.0;
            "GDB_TeachPoints".aPoints["GDB_TeachCmd".i16_SlotIdx].position[1] := 0.0;
            "GDB_TeachPoints".aPoints["GDB_TeachCmd".i16_SlotIdx].position[2] := 0.0;
            "GDB_TeachPoints".aPoints["GDB_TeachCmd".i16_SlotIdx].position[3] := 0.0;
            "GDB_TeachPoints".aPoints["GDB_TeachCmd".i16_SlotIdx].position[4] := 0.0;
            "GDB_TeachPoints".aPoints["GDB_TeachCmd".i16_SlotIdx].position[5] := 0.0;
            "GDB_TeachPoints".aJointAngles["GDB_TeachCmd".i16_SlotIdx, 1] := 0.0;
            "GDB_TeachPoints".aJointAngles["GDB_TeachCmd".i16_SlotIdx, 2] := 0.0;
            "GDB_TeachPoints".aJointAngles["GDB_TeachCmd".i16_SlotIdx, 3] := 0.0;
            "GDB_TeachPoints".aJointAngles["GDB_TeachCmd".i16_SlotIdx, 4] := 0.0;
            "GDB_TeachPoints".abCaptured["GDB_TeachCmd".i16_SlotIdx] := FALSE;
            "GDB_TeachCmd".i16_TeachStep := 30;
        ELSIF "GDB_TeachCmd".i16_TeachStep = 30 THEN
            "GDB_TeachCmd".i16_TeachStep := 0;
        END_IF;

        // --- Clear ALL slots (V1.1: zero BOTH TCP and joint arrays) ---
        IF #sRTRIG_ClearAll.Q AND #statTeachOK THEN
            FOR #i := 1 TO 16 DO
                "GDB_TeachPoints".aPoints[#i].position[0] := 0.0;
                "GDB_TeachPoints".aPoints[#i].position[1] := 0.0;
                "GDB_TeachPoints".aPoints[#i].position[2] := 0.0;
                "GDB_TeachPoints".aPoints[#i].position[3] := 0.0;
                "GDB_TeachPoints".aPoints[#i].position[4] := 0.0;
                "GDB_TeachPoints".aPoints[#i].position[5] := 0.0;
                "GDB_TeachPoints".aJointAngles[#i, 1] := 0.0;
                "GDB_TeachPoints".aJointAngles[#i, 2] := 0.0;
                "GDB_TeachPoints".aJointAngles[#i, 3] := 0.0;
                "GDB_TeachPoints".aJointAngles[#i, 4] := 0.0;
                "GDB_TeachPoints".abCaptured[#i] := FALSE;
            END_FOR;
            "GDB_TeachCmd".i16_TeachStep := 30;
        END_IF;
    END_REGION

    REGION Replay_FSM
        // Stop edge from any active state -> idle + abort move.
        IF #sRTRIG_StopReplay.Q AND #statTeachOK THEN
            IF "GDB_TeachCmd".i16_TeachStep >= 100 AND "GDB_TeachCmd".i16_TeachStep < 200 THEN
                "GDB_AxisCtrl".LKinCtrl.input.movelinear.bo_execute := FALSE;
                "GDB_TeachCmd".i16_TeachStep := 0;
                "GDB_TeachCmd".i16_ReplayIdx := 0;
            END_IF;
        END_IF;

        // Start edge -> seed FSM at LOAD_NEXT with idx=0 (so the first
        // increment lands on slot 1).
        IF #sRTRIG_StartReplay.Q AND #statTeachOK
                AND "GDB_TeachCmd".i16_TeachStep = 0
                AND "GDB_TeachPoints".i16_PointCount > 0 THEN
            "GDB_TeachCmd".bo_ReplayDone := FALSE;
            "GDB_TeachCmd".i16_ReplayIdx := 0;
            "GDB_TeachCmd".i16_TeachStep := 100;
        END_IF;

        // State 100: LOAD_NEXT -- scan forward from current idx+1 for
        // the next abCaptured slot. If none -> DONE (200).
        IF "GDB_TeachCmd".i16_TeachStep = 100 AND #statTeachOK THEN
            #tempReplayIdx := "GDB_TeachCmd".i16_ReplayIdx + 1;
            WHILE #tempReplayIdx <= 16 DO
                IF "GDB_TeachPoints".abCaptured[#tempReplayIdx] THEN
                    EXIT;
                END_IF;
                #tempReplayIdx := #tempReplayIdx + 1;
            END_WHILE;
            IF #tempReplayIdx > 16 THEN
                "GDB_TeachCmd".i16_TeachStep := 200;
            ELSE
                "GDB_TeachCmd".i16_ReplayIdx := #tempReplayIdx;
                "GDB_TeachCmd".i16_TeachStep := 110;
            END_IF;
        END_IF;

        // State 110: WRITE_TARGET -- copy slot to movelinear, pulse execute.
        IF "GDB_TeachCmd".i16_TeachStep = 110 AND #statTeachOK THEN
            "GDB_AxisCtrl".LKinCtrl.input.movelinear.targetposition.x := "GDB_TeachPoints".aPoints["GDB_TeachCmd".i16_ReplayIdx].position[0];
            "GDB_AxisCtrl".LKinCtrl.input.movelinear.targetposition.y := "GDB_TeachPoints".aPoints["GDB_TeachCmd".i16_ReplayIdx].position[1];
            "GDB_AxisCtrl".LKinCtrl.input.movelinear.targetposition.z := "GDB_TeachPoints".aPoints["GDB_TeachCmd".i16_ReplayIdx].position[2];
            "GDB_AxisCtrl".LKinCtrl.input.movelinear.targetposition.a := "GDB_TeachPoints".aPoints["GDB_TeachCmd".i16_ReplayIdx].position[3];
            "GDB_AxisCtrl".LKinCtrl.input.movelinear.targetposition.b := 0.0;
            "GDB_AxisCtrl".LKinCtrl.input.movelinear.targetposition.c := 0.0;
            "GDB_AxisCtrl".LKinCtrl.input.movelinear.r64_velocity     := "GDB_TeachCmd".lr_ReplayVel;
            "GDB_AxisCtrl".LKinCtrl.input.movelinear.r64_acceleration := 2000.0;
            "GDB_AxisCtrl".LKinCtrl.input.movelinear.r64_deceleration := 2000.0;
            "GDB_AxisCtrl".LKinCtrl.input.movelinear.r64_jerk         := 20000.0;
            "GDB_AxisCtrl".LKinCtrl.input.movelinear.bo_isPTP         := FALSE;
            "GDB_AxisCtrl".LKinCtrl.input.movelinear.bo_execute       := TRUE;
            "GDB_TeachCmd".i16_TeachStep := 120;
        END_IF;

        // State 120: WAIT_DONE -- poll for move-done edge, then advance.
        IF "GDB_TeachCmd".i16_TeachStep = 120 AND #statTeachOK
                AND #sRTRIG_MoveDone.Q THEN
            "GDB_AxisCtrl".LKinCtrl.input.movelinear.bo_execute := FALSE;
            "GDB_TeachCmd".i16_TeachStep := 100;  // load next captured slot
        END_IF;

        // State 200: REPLAY_DONE -- latch done, return to idle.
        IF "GDB_TeachCmd".i16_TeachStep = 200 AND #statTeachOK THEN
            "GDB_TeachCmd".bo_ReplayDone := TRUE;
            "GDB_TeachCmd".i16_ReplayIdx := 0;
            "GDB_TeachCmd".i16_TeachStep := 0;
        END_IF;
    END_REGION

    REGION Compute_PointCount
        // Count TRUE bits in abCaptured[1..16] each scan. Runs always
        // (NOT gated on statTeachOK) so HMI status display tracks even
        // when teach mode is off (e.g. operator inspects taught points
        // while in palletizing mode).
        #tempCount := 0;
        FOR #i := 1 TO 16 DO
            IF "GDB_TeachPoints".abCaptured[#i] THEN
                #tempCount := #tempCount + 1;
            END_IF;
        END_FOR;
        "GDB_TeachPoints".i16_PointCount := #tempCount;
    END_REGION

END_FUNCTION_BLOCK

FUNCTION_BLOCK "LKinCtrl_MC_JogFrame"
TITLE = LKinCtrl_MC_JogFrame
{ S7_Optimized_Access := 'TRUE' }
AUTHOR : 'handling.team.automation@siemens.com'
FAMILY : LKinCtrl
VERSION : 5.0
//Functionality: This function block provides various jog functionality for kinematics technology object.
   VAR_INPUT 
      jogForward : Bool := FALSE;   // Jog the kinematics forward in the selected jog direction
      jogBackward : Bool := FALSE;   // Jog the kinematics backward in the selected jog direction
      jogToPosition : Bool := FALSE;   // Jog the kinematics to the specified target position
      jogSPTP : Bool := FALSE;   // Jog the kinematics synchronous point to point
      jogDirection : USInt := 1;   // 1=x-direction, 2=y-direction, 3=z-direction, 4=a-direction, 5=b-direction, 6=c-direction, 7=Z-axis - about A,, 8=Y-axis - about B, 9=X-axis - about C
      jogModeInc : Bool := FALSE;   // 1=incremental jog mode, 0=continuous jog mode
      jogIncrement : LReal := 1.0;   // Specification of the jog increment
      targetPosition : "LKinCtrl_typeCartesianPosition";   // Specification of the target position
      coordSystem : DInt := 0;   // 0=WCS, 1= OCS1, 2=OCS2, 3=OCS3, 4=TCS, 100=MCS, 101=JCS
      linkconstellation : DWord := 16#FFFF_FFFF;   // Target joint position space
      turnJoint : Array[1..6] of DInt;   // Turn joint setting for move direct only
      tool : DInt := 1;   // 1= tool1, 2=tool2, 3=tool3
      dynamics : "LKinCtrl_typeDynamics";   // Specification of the jog dynamics
      userFrames { ExternalAccessible := 'False'; ExternalVisible := 'False'; ExternalWritable := 'False'} : Array["LKINCTRL_CS_NO_OF_FIRST_USER_FRAME".."LKINCTRL_CS_NO_OF_LAST_USER_FRAME"] of "LKinCtrl_typeFrame";
   END_VAR

   VAR_OUTPUT 
      done { ExternalWritable := 'False'} : Bool := FALSE;   // TRUE: Commanded functionality has been completed successfully
      busy { ExternalWritable := 'False'} : Bool := FALSE;   // TRUE: FB is not finished and new output values can be expected
      active { ExternalWritable := 'False'} : Bool := FALSE;   // TRUE: The setpoints are calculated
      error { ExternalWritable := 'False'} : Bool := FALSE;   // TRUE: An error occurred during the execution of the FB
      status { ExternalWritable := 'False'} : Word := #STATUS_NO_CALL;   // 16#0000 - 16#7FFF: Status of the FB, 16#8000 - 16#FFFF: Error identification
      remainingDistance { ExternalWritable := 'False'} : LReal := 0.0;   // Distance-to-go of the current job
      diagnostics { ExternalWritable := 'False'} : "LKinCtrl_typeJogFrameDiagnostics";   // Diagnostics information
   END_VAR

   VAR_IN_OUT 
      axesGroup {InstructionName := 'TO_Kinematics'; LibVersion := '9.0'} : TO_Kinematics;   // Kinematics technology object
   END_VAR

   VAR 
      instMC_SetTool {InstructionName := 'MC_SETTOOL'; LibVersion := '9.0'; ExternalAccessible := 'False'; ExternalVisible := 'False'; ExternalWritable := 'False'; S7_SetPoint := 'False'} : MC_SETTOOL;   // Instance MC_SetTool
      instMC_GroupStop {InstructionName := 'MC_GROUPSTOP'; LibVersion := '9.0'; ExternalAccessible := 'False'; ExternalVisible := 'False'; ExternalWritable := 'False'; S7_SetPoint := 'False'} : MC_GROUPSTOP;   // Instance MC_GroupStop
      instMC_MoveLinearAbsolute {InstructionName := 'MC_MOVELINEARABSOLUTE'; LibVersion := '9.0'; ExternalAccessible := 'False'; ExternalVisible := 'False'; ExternalWritable := 'False'; S7_SetPoint := 'False'} : MC_MOVELINEARABSOLUTE;   // Instance MC_MoveLinearAbsolute
      instMC_MoveLinearRelative {InstructionName := 'MC_MOVELINEARRELATIVE'; LibVersion := '9.0'; ExternalAccessible := 'False'; ExternalVisible := 'False'; ExternalWritable := 'False'; S7_SetPoint := 'False'} : MC_MOVELINEARRELATIVE;   // Instance MC_MoveLinearRelative
      instMC_MoveDirectAbsolute {InstructionName := 'MC_MOVEDIRECTABSOLUTE'; LibVersion := '9.0'; ExternalAccessible := 'False'; ExternalVisible := 'False'; ExternalWritable := 'False'; S7_SetPoint := 'False'} : MC_MOVEDIRECTABSOLUTE;   // Instance MC_MoveDirectAbsolute
      instMC_MoveDirectRelative {InstructionName := 'MC_MOVEDIRECTRELATIVE'; LibVersion := '9.0'; ExternalAccessible := 'False'; ExternalVisible := 'False'; ExternalWritable := 'False'; S7_SetPoint := 'False'} : MC_MOVEDIRECTRELATIVE;   // Instance MC_MoveDirectAbsolute
      statDone { ExternalAccessible := 'False'; ExternalVisible := 'False'; ExternalWritable := 'False'} : Bool := FALSE;   // Static value for output 'done'
      statBusy { ExternalAccessible := 'False'; ExternalVisible := 'False'; ExternalWritable := 'False'} : Bool := FALSE;   // Static value for output 'busy'
      statActive { ExternalAccessible := 'False'; ExternalVisible := 'False'; ExternalWritable := 'False'} : Bool := FALSE;   // Static value for output 'active'
      statError { ExternalAccessible := 'False'; ExternalVisible := 'False'; ExternalWritable := 'False'} : Bool := FALSE;   // Static value for output 'error'
      statStatus { ExternalAccessible := 'False'; ExternalVisible := 'False'; ExternalWritable := 'False'} : Word := #STATUS_NO_CALL;   // 0000=STATUS_EXECUTION_FINISHED; 7000=STATUS_NO_CALL; 7001=STATUS_FIRST_CALL; 7002=STATUS_SUBSEQUENT_CALL; 8600=ERR_UNDEFINED_STATE
      statRemainingDistance { ExternalAccessible := 'False'; ExternalVisible := 'False'; ExternalWritable := 'False'} : LReal := 0.0;   // Static value for remaining distance
      statFBState { ExternalAccessible := 'False'; ExternalVisible := 'False'; ExternalWritable := 'False'} : DInt := #FB_STATE_NO_PROCESSING;   // 0= NO PROCESSING; 10=IDLE; 20=SET_TOOL; 30=SET_DYNAMICS, 50=EXECUTE_MOVEMENT; 100=STOP
      statToolOld { ExternalAccessible := 'False'; ExternalVisible := 'False'; ExternalWritable := 'False'} : DInt := 1;   // Static value for tool
      statJogForwardOld { ExternalAccessible := 'False'; ExternalVisible := 'False'; ExternalWritable := 'False'} : Bool := FALSE;   // Static value for jog forward command
      statJogBackwardOld { ExternalAccessible := 'False'; ExternalVisible := 'False'; ExternalWritable := 'False'} : Bool := FALSE;   // Static value for jog backward command
      statJogToPositionOld { ExternalAccessible := 'False'; ExternalVisible := 'False'; ExternalWritable := 'False'} : Bool := FALSE;   // Static value for jog to position command
      statJogSPTPOld { ExternalAccessible := 'False'; ExternalVisible := 'False'; ExternalWritable := 'False'} : Bool := FALSE;   // Static value for jog sPTP command
      statOrientationDynamicsChanged { ExternalAccessible := 'False'; ExternalVisible := 'False'; ExternalWritable := 'False'} : Bool := FALSE;   // Static value indicates that default orientation dynamics have been changed
      statOrientationDynamicsOld { ExternalAccessible := 'False'; ExternalVisible := 'False'; ExternalWritable := 'False'; S7_SetPoint := 'False'} : "LKinCtrl_typePathDynamics";   // Static value for orientation dynamics
      statRotMatrix1 { ExternalAccessible := 'False'; ExternalVisible := 'False'; ExternalWritable := 'False'} : Array[1..3, 1..3] of LReal;   // Rotationmatrix 1
      statRotMatrix2 { ExternalAccessible := 'False'; ExternalVisible := 'False'; ExternalWritable := 'False'} : Array[1..3, 1..3] of LReal;   // Rotationmatrix 2
      statRotMatrix3 { ExternalAccessible := 'False'; ExternalVisible := 'False'; ExternalWritable := 'False'} : Array[1..3, 1..3] of LReal;   // Rotationmatrix 3
      statTypeOfKinematics { ExternalAccessible := 'False'; ExternalVisible := 'False'; ExternalWritable := 'False'} : DInt;   // Static value to store type of kinematics
      statTypeOfKinematicsOld { ExternalAccessible := 'False'; ExternalVisible := 'False'; ExternalWritable := 'False'} : DInt;   // Static value to detect change of kinematics type
      statFrameCoordinateConfigurable { ExternalAccessible := 'False'; ExternalVisible := 'False'; ExternalWritable := 'False'} : Array[1..6] of Bool;   // Static array showing which DOF are available
      statUpperFrameLimit { ExternalAccessible := 'False'; ExternalVisible := 'False'; ExternalWritable := 'False'} : Array[1..6] of LReal;   // Static array with upper limits for positions
      statLowerFrameLimit { ExternalAccessible := 'False'; ExternalVisible := 'False'; ExternalWritable := 'False'} : Array[1..6] of LReal;   // Static array with lower limits for positions
      stat5D6D { ExternalAccessible := 'False'; ExternalVisible := 'False'; ExternalWritable := 'False'} : Bool;   // Static variable, TRUE. 5D/6D, FALSE < 5D
      statStatusBeforeResetTool { ExternalAccessible := 'False'; ExternalVisible := 'False'; ExternalWritable := 'False'} : Word;   // Status saved before reset tool state
   END_VAR

   VAR_TEMP 
      tempJogForward : Bool;   // Temporary variable for jog forward input
      tempJogBackward : Bool;   // Temporary variable for jog backward input
      tempJogToPosition : Bool;   // Temporary variable for jog to position input
      tempJogSPTP : Bool;   // Temporary variable for jog sptp input
      tempCounter : DInt;   // Temporary variable for counter
      tempRet : Int;   // Temporary variable for time stamp if error occurred
      tempJogDistance : LReal;   // Temporary variable for jog distance
      tempError : Bool;   // Temporary variable for error in subfunction
      tempRetStatus : Word;   // Temporary variable for return value of subfunction
      tempDirectionOk : Bool;   // Temporary variable to check if jog direction is ok
      tempCoordSystemOk : Bool;   // Temporary variable to check if coordinate system is ok
      tempDistToLimit : LReal;   // Temporary variable to calculate distance to joint limit
      tempOk : Bool;   // Temporary variable to check if condition is ok
      tempLimitJCS : LReal;   // Temporary variable for JCS limit
      tempLimitMCS : LReal;   // Termporary variable for MCS limit
      tempDistToLimitJCS : LReal;   // Temporary variable for distance to JCS limit
      tempDistToLimitMCS : LReal;   // Temporary variable for distance to MCS limit
      tempDistToLimitACJCS : LReal;   // Temporary variable for distance to JCS limit of affected axes
      tempDistToLimitACMCS : LReal;   // Temporary variable for distance to MCS limit of affected axes
      tempDistToLimitACMin : LReal;   // Temporary variable for minimum distance to limit of affected axes
      tempLimitACJCS : LReal;   // Temporary variable for effective joint limit
      tempLimitACMCS : LReal;   // Temporary variable for effective joint limit
      tempFactor : LReal;   // Temporary variable for coupling factor
      tempCausingAxis : UDInt;   // Temporary variable for causing axis
      tempAffectedAxis : DInt;   // Temporary variable for affected axis
      tempAxisPosition : Array[1..#NO_OF_AXES] of LReal;   // Temporary variable for axis positions
      tempJointPosition : Array[1..#NO_OF_AXES] of LReal;   // Temporary variable for joint positions
      tempJointUpperLimit : Array[1..#NO_OF_AXES] of LReal;   // Temporary variable for joint upper limit
      tempJointLowerLimit : Array[1..#NO_OF_AXES] of LReal;   // Temporary variable for joint lower limit
      tempAxisSWLimitActive : Array[1..#NO_OF_AXES] of Bool;   // Temporary variable for axis SW limit active
      tempAxisSWLimitMaxPos : Array[1..#NO_OF_AXES] of LReal;   // Temporary variable for axis SW limit max. position
      tempAxisSWLimitMinPos : Array[1..#NO_OF_AXES] of LReal;   // Temporary variable for axis SW limit min. position
      tempTcpInUcs : Array[1..#NO_OF_AXES] of LReal;
      tempRefPosAxis {InstructionName := 'TO_PositioningAxis'; LibVersion := '9.0'} : REF_TO TO_PositioningAxis;   // Reference to position axis
   END_VAR

   VAR CONSTANT 
      FB_STATE_NO_PROCESSING : DInt := 0;   // FB state: No processing
      FB_STATE_CMD_CONFIGURATION : DInt := 10;   // FB state: Basic command configuration are set depending on input parameter
      FB_STATE_SET_TOOL : DInt := 20;   // FB state: Tool change is performed if required
      FB_STATE_EXECUTE_MOVEMENT : DInt := 50;   // FB state: Command is being executed
      FB_STATE_RESET_TOOL : DInt := 60;
      FB_STATE_STOP : DInt := 100;   // FB state: Kinematics movement is stopped
      STATUS_EXECUTION_FINISHED : Word := 16#0000;   // The command execution is finished by reaching the target position or stopping the jog command
      STATUS_NO_CALL : Word := 16#7000;   // No call of FB
      STATUS_FIRST_CALL : Word := 16#7001;   // First cycle of FB after enabling
      STATUS_SUBSEQUENT_CALL : Word := 16#7002;   // FB enabled
      STATUS_OUT_OF_SW_LIMIT_BOUNDARIES : Word := 16#7010;   // Warning - out of axis software limits
      STATUS_OUT_OF_JOINT_LIMITS : Word := 16#7011;   // Warning - out of joint limits (Kin 5D/6D)
      ERR_UNDEFINED_STATE : Word := 16#8600;   // Error due to an undefined FB state
      ERR_TO_KINEMATICS : Word := 16#8001;   // Error at technology object kinematics
      ERR_INVALID_JOG_DIRECTION : Word := 16#8007;   // The specified jog direction is invalid (valid are: 1=x-direction, 2=y-direction, 3=z-direction, 4=a-direction, 5=b-direction, 6=c-direction, 7=Z-axis - about A,, 8=Y-axis - about B, 9=X-axis - about C)
      ERR_MOTION_JOB_IN_PROGRESS : Word := 16#8090;   // A motion job is in progress or the kinematics control panel is activated
      ERR_TWO_JOG_COMMANDS_SIMULTANEOUSLY : Word := 16#8091;   // Two jog commands were triggered simultaneously
      ERR_INVALID_COORDINATE_SYSTEM : Word := 16#80B1;   // The specified coordinate system is invalid (valid values are 0=WCS, 1= OCS1, 2=OCS2, 3=OCS3)
      ERR_INVALID_TOOL : Word := 16#80CA;   // The specified tool is invalid (valid values are 1= tool1, 2=tool2, 3=tool3)
      ERR_JOG_DIRECTION_NOT_POSSIBLE : Word := 16#8100;   // The specified jog direction is not possible due to reduced degrees of freedom (5D)
      MAX_DISTANCE : LReal := 70000.0;   // The value is set for relative linear movement as jog increment for icremental jog mode
      MAX_DISTANCE_ROTATION : LReal := 1000.0;   // The value is set for absolute linear movement as distance in TCS
      L_BOUND_TOOL : DInt := 1;   // Lower bound for tool selection
      U_BOUND_TOOL : DInt := 3;   // Upper bound for tool selection
      L_BOUND_JOG_DIRECTION : DInt := 1;   // Lower bound for jog direction selection
      U_BOUND_JOG_DIRECTION : DInt := 9;   // Upper bound for jog direction selection
      L_BOUND_COORDSYSTEM : DInt := 0;   // Lower bound for coordinate system selection
      U_BOUND_COORDSYSTEM : DInt := 4;   // Upper bound for coordinate system selection
      INDEX_COORDSYSTEM_MCS : DInt := 100;   // Coordinate system index for MCS
      INDEX_COORDSYSTEM_JCS : DInt := 101;   // Coordinate system index for JCS
      INDEX_COORDSYSTEM_TCS : DInt := 4;   // Coordinate system index for TCS
      JOG_DIRECTION_X : USInt := 1;   // Jog direction index for X
      JOG_DIRECTION_Y : USInt := 2;   // Jog direction index for Y
      JOG_DIRECTION_Z : USInt := 3;   // Jog direction index for Z
      JOG_DIRECTION_A : USInt := 4;   // Jog direction index for A
      JOG_DIRECTION_B : USInt := 5;   // Jog direction index for B
      JOG_DIRECTION_C : USInt := 6;   // Jog direction index for C
      JOG_DIRECTION_RZ : USInt := 7;   // Jog direction index for RZ
      JOG_DIRECTION_RY : USInt := 8;   // Jog direction index for RY
      JOG_DIRECTION_RX : USInt := 9;   // Jog direction index for RX
      TOLERANCE_C : LReal := 0.01;   // Tolerance for target position C for 5D Kinematics
      NO_OF_AXES : DInt := 6;   // Number of available axes
      NO_OF_COUPLINGS : DInt := 5;   // Number of available axes couplings
      SAFETY_DISTANCE : LReal := 0.1;   // Safety distance to limit of axes (Joint limit and software limit switch)
      MOTION_TYPE_LINEAR : DInt := 0;
      MOTION_TYPE_ROTARY : DInt := 1;
   END_VAR


BEGIN
	//=============================================================================
	// SIEMENS AG
	// (c)Copyright 2018 All Rights Reserved
	//-----------------------------------------------------------------------------
	// Library:       LKinCtrl
	// Tested with:   S7-1516T
	// Engineering:   TIA Portal V15
	// Restrictions:  -
	// Requirements:  S7-1500T FW 2.5
	// Functionality: LKinCtrl_MC_JogFrame
	// This function block provides various jog functionality for kinematics technology object
	//
	// Support: tech.team.motioncontrol@siemens.com
	// Note: Parameter comments are only available in language 'English (United States)'
	//-----------------------------------------------------------------------------
	// Change log table:
	// Version  Date        Expert in charge   Changes applied
	// 01.00.00 05.04.2018  IP                 First released version
	// 01.00.01 24.04.2018  IP                 Hotfix - initialization - no functional changes
	// 01.01.00 31.07.2018  IP                 Adjustment of input validation
	//                                         New wait condition for next movement until stopping is done
	//                                         Additional output parameter active and remaining distance
	// 01.01.01 07.08.2018  IP                 Hotfix - constant MAX_DISTANCE decreased
	// 01.01.02 09.01.2019  IP                 Hotfix - error indification adjusted
	// 01.01.03 14.01.2019  IP                 Hotfix - dynamics configuration adjusted
	// 01.01.04 12.07.2021  FF                 Added Synchronous point to point jogging
	// 01.01.05 14.12.2021  FR                 Fix for orientation dynamics and refactor
	// 01.01.06 15.07.2022  FR                 Fix for Override = 0 and fast toggle of inputs
	// 02.00.00 18.01.2023  FR                 Updated to 6 axis
	// 02.00.01 15.03.2023  FR                 Bugfix for 2D kinematics
	// 02.00.02 02.05.2024  FR                 Check for 5D jogging -> New error 16#8100
	// 02.01.00 05.09.2024  FR                 Reset tool after jog
	// 02.02.00 10.09.2024  JH                 Added UCS jogging
	//=============================================================================
	
	#tempJogForward := #jogForward; // Work with temporary value / create process image
	#tempJogBackward := #jogBackward;
	#tempJogToPosition := #jogToPosition;
	#tempJogSPTP := #jogSPTP;
	
	REGION TRIGGERING
	  IF ((#tempJogForward AND NOT #statJogForwardOld) // Check if FB is triggered
	    OR (#tempJogBackward AND NOT #statJogBackwardOld)
	    OR (#tempJogToPosition AND NOT #statJogToPositionOld)
	    OR (#tempJogSPTP AND NOT #statJogSPTPOld))
	    AND (#statStatus = #STATUS_NO_CALL)
	    AND (#statFBState = #FB_STATE_NO_PROCESSING)
	  THEN
	    // First call; set FB variables for outputs
	    #statBusy := TRUE;
	    #statDone := FALSE;
	    #statActive := FALSE;
	    #statError := FALSE;
	    #statRemainingDistance := 0.0;
	    #statStatus := #STATUS_FIRST_CALL;
	    // Get type of kinematics
	    #statTypeOfKinematics := #axesGroup.Kinematics.TypeOfKinematics;
	    
	    // check if kinematics is 4D or more
	    CASE #statTypeOfKinematics OF
	      26, 27, // 3D + A,B
	      25, 36: // 3D + A,B,C
	        #stat5D6D := TRUE;
	      ELSE
	        // Reset variable
	        #stat5D6D := FALSE;
	    END_CASE;
	    
	    IF #statTypeOfKinematicsOld <> #statTypeOfKinematics THEN
	      "LKinCtrl_FramesValidValues"(mode                        := 0, // Positions
	                                   typeOfKinematics            := #statTypeOfKinematics,
	                                   frameCoordinateConfigurable => #statFrameCoordinateConfigurable,
	                                   upperLimitFrame             => #statUpperFrameLimit,
	                                   lowerLimitFrame             => #statLowerFrameLimit);
	      #statTypeOfKinematicsOld := #statTypeOfKinematics;
	    END_IF;
	    
	    CASE #statTypeOfKinematics OF
	      1, 5, 11, 15, 31,  // 2D kinematics
	      2, 6, 12, 16, 20, 32:  // 2D + orientation axis A
	        IF #coordSystem = #INDEX_COORDSYSTEM_MCS OR #coordSystem = #INDEX_COORDSYSTEM_JCS THEN
	          // Allow A2 but not A3
	          #statFrameCoordinateConfigurable[2] := TRUE;
	          #statFrameCoordinateConfigurable[3] := FALSE;
	        ELSE
	          // Allow Z but not Y
	          #statFrameCoordinateConfigurable[2] := FALSE;
	          #statFrameCoordinateConfigurable[3] := TRUE;
	        END_IF;
	    END_CASE;
	    
	    // Check jog direction
	    IF #tempJogToPosition OR #tempJogSPTP THEN
	      #tempDirectionOk := TRUE; // direction is not used
	    ELSE
	      CASE #jogDirection OF
	        #JOG_DIRECTION_X..#JOG_DIRECTION_C:
	          #tempDirectionOk := #statFrameCoordinateConfigurable[#jogDirection];
	        ELSE
	          ;
	      END_CASE;
	      
	      // Special cases for RZ,RY,RX (5D/6D)
	      CASE #statTypeOfKinematics OF
	        26, 27: // 3D + A,B
	          #tempDirectionOk := (#jogDirection >= #L_BOUND_JOG_DIRECTION AND #jogDirection <= #U_BOUND_JOG_DIRECTION)
	          AND NOT (#jogDirection = #JOG_DIRECTION_C);
	          
	        25, 36: // 3D + A,B,C
	          #tempDirectionOk := #jogDirection >= #L_BOUND_JOG_DIRECTION AND #jogDirection <= #U_BOUND_JOG_DIRECTION;
	        ELSE
	          ;
	      END_CASE;
	      
	      // No linear jog in cartesian allowed for Scara 2D+A but MCS/JCS is ok
	      IF (#statTypeOfKinematics = 20) AND (#coordSystem <> #INDEX_COORDSYSTEM_MCS) AND (#coordSystem <> #INDEX_COORDSYSTEM_JCS) THEN
	        #tempDirectionOk := FALSE;
	      END_IF;
	    END_IF;
	    
	    // Check coordinate system
	    CASE #coordSystem OF
	      "CS_WCS".."CS_OCS3":
	        #tempCoordSystemOk := TRUE; // always true?
	        
	      "LKINCTRL_CS_NO_OF_FIRST_USER_FRAME".. "LKINCTRL_CS_NO_OF_LAST_USER_FRAME":
	        #tempCoordSystemOk := TRUE; // always true?
	        
	      #INDEX_COORDSYSTEM_MCS:
	        #tempCoordSystemOk := (#tempJogToPosition = FALSE); // Linear not allowed
	        
	        // Do not allow jogDirection 7..9
	        IF #jogDirection >= #JOG_DIRECTION_RZ THEN
	          #tempDirectionOk := FALSE;
	        END_IF;
	        
	      #INDEX_COORDSYSTEM_JCS:
	        #tempCoordSystemOk := (#tempJogToPosition = FALSE AND #stat5D6D = TRUE); // Not Linear and atleast 5D
	        
	        // Do not allow jogDirection 7..9
	        IF #jogDirection >= #JOG_DIRECTION_RZ THEN
	          #tempDirectionOk := FALSE;
	        END_IF;
	        
	      #INDEX_COORDSYSTEM_TCS:
	        #tempCoordSystemOk := (#tempJogSPTP = FALSE); // SPTP not possible in TCS
	        
	      ELSE
	        // Invalid coordinate system
	        #tempCoordSystemOk := FALSE;
	    END_CASE;
	    
	    IF #tempDirectionOk = FALSE THEN
	      #statStatus := #ERR_INVALID_JOG_DIRECTION;
	    ELSIF #tool < #L_BOUND_TOOL OR #tool > #U_BOUND_TOOL THEN // check tool
	      #statStatus := #ERR_INVALID_TOOL;
	    ELSIF #tempCoordSystemOk = FALSE THEN
	      #statStatus := #ERR_INVALID_COORDINATE_SYSTEM;
	    ELSIF NOT #axesGroup.StatusWord.%X6 THEN // check if a motion job is in progress or the kinematics control panel is activated
	      #statStatus := #ERR_MOTION_JOB_IN_PROGRESS;
	    ELSE // all input parameter are valid     
	      
	      // reset execute inputs
	      #instMC_GroupStop.Execute := FALSE;
	      #instMC_MoveLinearAbsolute.Execute := FALSE;
	      #instMC_MoveLinearRelative.Execute := FALSE;
	      #instMC_MoveDirectAbsolute.Execute := FALSE;
	      #instMC_MoveDirectRelative.Execute := FALSE;
	      #instMC_SetTool.Execute := FALSE;
	      
	      // call FBs with execute = false
	      #instMC_GroupStop(AxesGroup := #axesGroup);
	      #instMC_MoveLinearAbsolute(AxesGroup := #axesGroup);
	      #instMC_MoveLinearRelative(AxesGroup := #axesGroup);
	      #instMC_MoveDirectAbsolute(AxesGroup := #axesGroup);
	      #instMC_MoveDirectRelative(AxesGroup := #axesGroup);
	      #instMC_SetTool(AxesGroup := #axesGroup);
	      
	      // get actual tool number
	      #statToolOld := #axesGroup.StatusTool.ActiveTool;
	      
	      // safe default dynamics for orientation axis
	      #statOrientationDynamicsOld.velocity := #axesGroup.DynamicDefaults.Orientation.Velocity;
	      #statOrientationDynamicsOld.acceleration := #axesGroup.DynamicDefaults.Orientation.Acceleration;
	      #statOrientationDynamicsOld.deceleration := #axesGroup.DynamicDefaults.Orientation.Deceleration;
	      #statOrientationDynamicsOld.jerk := #axesGroup.DynamicDefaults.Orientation.Jerk;
	      #statOrientationDynamicsChanged := FALSE;
	      
	      // state machine - start functionality
	      #statFBState := #FB_STATE_CMD_CONFIGURATION;
	    END_IF;
	    
	  ELSIF (#statStatus = #STATUS_FIRST_CALL) THEN
	    #statStatus := #STATUS_SUBSEQUENT_CALL;
	  END_IF;
	  
	END_REGION TRIGGERING
	
	IF (#statStatus = #STATUS_NO_CALL) THEN // Nothing to do -> End here to reduce "system load"
	  RETURN;
	END_IF;
	
	REGION STOP_MOTION
	  // detection of falling edge on jog command
	  IF ((NOT #tempJogForward AND #statJogForwardOld)
	    OR (NOT #tempJogBackward AND #statJogBackwardOld)
	    OR (NOT #tempJogToPosition AND #statJogToPositionOld)
	    OR (NOT #tempJogSPTP AND #statJogSPTPOld))
	    AND NOT (#statFBState = #FB_STATE_NO_PROCESSING)
	  THEN // stop jog command
	    #statFBState := #FB_STATE_STOP;
	    
	    // two jog commands simultaneously    
	  ELSIF ((#tempJogBackward AND #tempJogForward)
	    OR (#tempJogBackward AND #tempJogToPosition)
	    OR (#tempJogBackward AND #tempJogSPTP)
	    OR (#tempJogForward AND #tempJogToPosition)
	    OR (#tempJogForward AND #tempJogSPTP)
	    OR (#tempJogToPosition AND #tempJogSPTP))
	    AND NOT (#statFBState = #FB_STATE_NO_PROCESSING)
	  THEN // stop jog command
	    #statFBState := #FB_STATE_STOP;
	    #statStatus := #ERR_TWO_JOG_COMMANDS_SIMULTANEOUSLY;
	  END_IF;
	  
	  IF #statStatus <> #STATUS_FIRST_CALL
	    AND (#statStatus.%X15 = FALSE)
	  THEN
	    IF #axesGroup.StatusWord.%X1 // general TO error
	      OR #instMC_MoveLinearAbsolute.Error
	      OR #instMC_MoveLinearRelative.Error
	      OR #instMC_MoveDirectAbsolute.Error
	      OR #instMC_MoveDirectRelative.Error
	      OR #instMC_GroupStop.Error
	      OR (#instMC_SetTool.Error AND NOT (#statFBState = #FB_STATE_RESET_TOOL))
	    THEN
	      #statFBState := #FB_STATE_STOP;
	    END_IF;
	  END_IF;
	END_REGION
	
	// Edge detection 'execute' input
	#statJogForwardOld := #tempJogForward;
	#statJogBackwardOld := #tempJogBackward;
	#statJogToPositionOld := #tempJogToPosition;
	#statJogSPTPOld := #tempJogSPTP;
	
	REGION RESET_DEFAULT_ORIENTATION_DYNAMICS
	  IF (#instMC_MoveLinearRelative.Busy OR #instMC_MoveLinearAbsolute.Busy OR #statFBState = #FB_STATE_STOP)
	    AND #statOrientationDynamicsChanged
	  THEN // reset default orientation dynamics
	    #axesGroup.DynamicDefaults.Orientation.Velocity := #statOrientationDynamicsOld.velocity;
	    #axesGroup.DynamicDefaults.Orientation.Acceleration := #statOrientationDynamicsOld.acceleration;
	    #axesGroup.DynamicDefaults.Orientation.Deceleration := #statOrientationDynamicsOld.deceleration;
	    #axesGroup.DynamicDefaults.Orientation.Jerk := #statOrientationDynamicsOld.jerk;
	    #statOrientationDynamicsChanged := FALSE;
	  END_IF;
	END_REGION
	
	REGION ACTIVE_OUTPUT
	  // set active output if any of motion commands is active
	  #statActive := #instMC_MoveLinearAbsolute.Active
	  OR #instMC_MoveLinearRelative.Active
	  OR #instMC_MoveDirectAbsolute.Active
	  OR #instMC_MoveDirectRelative.Active
	  OR #instMC_GroupStop.Active;
	END_REGION
	
	REGION REMAINING_DISTANCE
	  // set remaining distance at output if incremental mode active or while jogging to target position
	  IF #instMC_MoveLinearAbsolute.Busy THEN
	    #statRemainingDistance := #instMC_MoveLinearAbsolute.RemainingDistance;
	  ELSIF #instMC_MoveLinearRelative.Busy AND #jogModeInc THEN
	    #statRemainingDistance := #instMC_MoveLinearRelative.RemainingDistance;
	  ELSE
	    #statRemainingDistance := 0.0;
	  END_IF;
	END_REGION
	
	REGION STATE_MACHINE
	  CASE #statFBState OF // State machine of FB
	    #FB_STATE_NO_PROCESSING: // No processing active (Note: this state must always be present and left empty)
	      ;
	      
	    #FB_STATE_CMD_CONFIGURATION:
	      // Check for override <> 0 -> Only execute commands if override <> 0 as there are issues with TO_Kin if override = 0
	      IF #axesGroup.Override.Velocity <> 0 THEN
	        REGION CONFIGURATION
	          // jog forward or backward
	          //*********************************************************************************************************
	          IF #tempJogForward OR #tempJogBackward THEN
	            REGION JOG
	            // jog distance + dynamic adaption
	            IF #jogModeInc THEN // incremental
	              #tempJogDistance := #jogIncrement;
	              #instMC_MoveLinearAbsolute.DynamicAdaption := "DA_WITH_VARIABLE_LIMITS";
	              #instMC_MoveLinearRelative.DynamicAdaption := "DA_WITH_VARIABLE_LIMITS";
	            ELSE // continouos
	              // switch off dynamic adaption for continouos mode
	              #instMC_MoveLinearAbsolute.DynamicAdaption := "DA_DEACTIVATED";//"DA_WITH_VARIABLE_LIMITS";
	              #instMC_MoveLinearRelative.DynamicAdaption := "DA_DEACTIVATED";//"DA_WITH_VARIABLE_LIMITS";
	              // Check direction
	              IF #coordSystem = #INDEX_COORDSYSTEM_MCS OR #coordSystem = #INDEX_COORDSYSTEM_JCS THEN
	                CASE #jogDirection OF
	                  1:
	                    #tempRefPosAxis ?= #axesGroup.KinematicsAxis.A1;
	                  2:
	                    #tempRefPosAxis ?= #axesGroup.KinematicsAxis.A2;
	                  3:
	                    #tempRefPosAxis ?= #axesGroup.KinematicsAxis.A3;
	                  4:
	                    #tempRefPosAxis ?= #axesGroup.KinematicsAxis.A4;
	                  5:
	                    #tempRefPosAxis ?= #axesGroup.KinematicsAxis.A5;
	                  6:
	                    #tempRefPosAxis ?= #axesGroup.KinematicsAxis.A6;
	                END_CASE;
	                IF #tempRefPosAxis <> NULL THEN
	                  IF #tempRefPosAxis^.Properties.MotionType = #MOTION_TYPE_LINEAR THEN
	                    #tempJogDistance := #MAX_DISTANCE;
	                  ELSE
	                    #tempJogDistance := #MAX_DISTANCE_ROTATION;
	                  END_IF;
	                END_IF;
	              ELSE // cartesian jogging
	                IF #jogDirection < #JOG_DIRECTION_A THEN
	                  #tempJogDistance := #MAX_DISTANCE;
	                ELSE
	                  #tempJogDistance := #MAX_DISTANCE_ROTATION;
	                END_IF;
	              END_IF;
	            END_IF;
	            
	            // invert distance if backward
	            IF #tempJogBackward THEN
	              #tempJogDistance *= -1;
	            END_IF;
	            
	            CASE #jogDirection OF
	              #JOG_DIRECTION_X..#JOG_DIRECTION_C:
	                IF #coordSystem = #INDEX_COORDSYSTEM_MCS OR #coordSystem = #INDEX_COORDSYSTEM_JCS THEN
	                  // set MC_MoveDirectRelative parameter
	                  #instMC_MoveDirectRelative.CoordSystem := #coordSystem;
	                  #instMC_MoveDirectRelative.VelocityFactor := #dynamics.sPTP.velocityFactor;
	                  #instMC_MoveDirectRelative.AccelerationFactor := #dynamics.sPTP.accelerationFactor;
	                  #instMC_MoveDirectRelative.DecelerationFactor := #dynamics.sPTP.decelerationFactor;
	                  #instMC_MoveDirectRelative.JerkFactor := #dynamics.sPTP.jerkFactor;
	                  #instMC_MoveDirectRelative.LinkConstellation := #linkconstellation;
	                  #instMC_MoveDirectRelative.TurnJoint := #turnJoint;
	                  
	                  // initialize jog distance - clear old values
	                  FOR #tempCounter := 1 TO 6 DO
	                    #instMC_MoveDirectRelative.Distance[#tempCounter] := 0.0;
	                  END_FOR;
	                  
	                  // MCS / JCS
	                  FOR #tempCounter := 1 TO #NO_OF_AXES DO
	                    #tempAxisPosition[#tempCounter] := #axesGroup.AxesData.A[#tempCounter].Position;
	                    IF (#stat5D6D) THEN
	                      #tempJointPosition[#tempCounter] := #axesGroup.JointData.J[#tempCounter].Position;
	                    END_IF;
	                  END_FOR;
	                  
	                  // Check if jointalready outside limits
	                  #tempOk := TRUE;
	                  IF (#stat5D6D) THEN
	                    FOR #tempCounter := 1 TO #NO_OF_AXES DO
	                      #tempJointUpperLimit[#tempCounter] := #axesGroup.Joint.J[#tempCounter].UpperLimit;
	                      #tempJointLowerLimit[#tempCounter] := #axesGroup.Joint.J[#tempCounter].LowerLimit;
	                      
	                      IF ((#tempJointPosition[#tempCounter] >= #tempJointUpperLimit[#tempCounter]) OR
	                        (#tempJointPosition[#tempCounter] <= #tempJointLowerLimit[#tempCounter]))
	                      THEN
	                        #tempOk := FALSE;
	                        #statStatus := #STATUS_OUT_OF_JOINT_LIMITS;
	                        EXIT; // Already outside joint limit
	                      ELSE
	                        // Take safety distance into account
	                        #tempJointUpperLimit[#tempCounter] -= #SAFETY_DISTANCE;
	                        #tempJointLowerLimit[#tempCounter] += #SAFETY_DISTANCE;
	                      END_IF;
	                    END_FOR;
	                  END_IF;
	                  
	                  // Check if axis is already outside limits
	                  IF (#tempOk) THEN
	                    FOR #tempCounter := 1 TO #NO_OF_AXES DO
	                      CASE #tempCounter OF
	                        1:
	                          #tempRefPosAxis ?= #axesGroup.KinematicsAxis.A1;
	                        2:
	                          #tempRefPosAxis ?= #axesGroup.KinematicsAxis.A2;
	                        3:
	                          #tempRefPosAxis ?= #axesGroup.KinematicsAxis.A3;
	                        4:
	                          #tempRefPosAxis ?= #axesGroup.KinematicsAxis.A4;
	                        5:
	                          #tempRefPosAxis ?= #axesGroup.KinematicsAxis.A5;
	                        6:
	                          #tempRefPosAxis ?= #axesGroup.KinematicsAxis.A6;
	                      END_CASE;
	                      
	                      IF (#tempRefPosAxis <> NULL) THEN
	                        #tempAxisSWLimitActive[#tempCounter] := #tempRefPosAxis^.PositionLimits_SW.Active;
	                        #tempAxisSWLimitMaxPos[#tempCounter] := #tempRefPosAxis^.PositionLimits_SW.MaxPosition - #SAFETY_DISTANCE;
	                        #tempAxisSWLimitMinPos[#tempCounter] := #tempRefPosAxis^.PositionLimits_SW.MinPosition + #SAFETY_DISTANCE;
	                      ELSE
	                        #tempAxisSWLimitActive[#tempCounter] := FALSE;
	                      END_IF;
	                    END_FOR;
	                  END_IF;
	                  
	                  IF (#tempOk) THEN
	                    IF (#tempJogForward) // Positive direction
	                    THEN
	                      // positive direction
	                      IF (#stat5D6D) THEN
	                        #tempLimitJCS := #tempJointUpperLimit[#jogDirection];
	                      END_IF;
	                      IF (#tempAxisSWLimitActive[#jogDirection]) THEN
	                        #tempLimitMCS := #tempAxisSWLimitMaxPos[#jogDirection];
	                      END_IF;
	                    ELSE
	                      // negative direction
	                      IF (#stat5D6D) THEN
	                        #tempLimitJCS := #tempJointLowerLimit[#jogDirection];
	                      END_IF;
	                      IF (#tempAxisSWLimitActive[#jogDirection]) THEN
	                        #tempLimitMCS := #tempAxisSWLimitMinPos[#jogDirection];
	                      END_IF;
	                    END_IF;
	                    
	                    IF (#stat5D6D) THEN
	                      #tempDistToLimitJCS := ABS(#tempLimitJCS - #tempJointPosition[#jogDirection]);
	                      IF #jogDirection < #JOG_DIRECTION_A THEN
	                        #tempDistToLimitACJCS := #MAX_DISTANCE;
	                      ELSE
	                        #tempDistToLimitACJCS := #MAX_DISTANCE_ROTATION;
	                      END_IF;
	                    ELSE
	                      #tempDistToLimitJCS := #MAX_DISTANCE;
	                    END_IF;
	                    
	                    IF (#tempAxisSWLimitActive[#jogDirection]) THEN
	                      #tempDistToLimitMCS := ABS(#tempLimitMCS - #tempAxisPosition[#jogDirection]);
	                    ELSE
	                      #tempDistToLimitMCS := #MAX_DISTANCE;
	                    END_IF;
	                    IF #jogDirection < #JOG_DIRECTION_A THEN
	                      #tempDistToLimitACMin := #MAX_DISTANCE;
	                    ELSE
	                      #tempDistToLimitACMin := #MAX_DISTANCE_ROTATION;
	                    END_IF;
	                    
	                    // Use smaller limit
	                    #tempDistToLimit := MIN(IN1 := #tempDistToLimitJCS, IN2 := #tempDistToLimitMCS, IN3 := ABS(#tempJogDistance));
	                    
	                    // Check if an axis coupling is present
	                    FOR #tempCounter := 1 TO #NO_OF_COUPLINGS DO
	                      IF (#axesGroup.AxisCoupling.N[#tempCounter].Enable = FALSE) THEN // Coupling not enabled
	                        CONTINUE;
	                      END_IF;
	                      
	                      #tempFactor := #axesGroup.AxisCoupling.N[#tempCounter].Factor; // Get factor
	                      
	                      IF (#tempFactor = 0.0) THEN // Check if factor is 0.0
	                        CONTINUE;
	                      END_IF;
	                      
	                      #tempCausingAxis := #axesGroup.AxisCoupling.N[#tempCounter].CausingAxis; // Get causing axis
	                      
	                      IF #tempCausingAxis <> #jogDirection THEN // Causing axis is not current direction
	                        CONTINUE;
	                      END_IF;
	                      
	                      #tempAffectedAxis := UDINT_TO_DINT(#axesGroup.AxisCoupling.N[#tempCounter].AffectedAxis); // Get affected axis
	                      
	                      // Calculate limit
	                      IF (((#tempFactor > 0) AND #tempJogForward) OR // Positive direction
	                        ((#tempFactor < 0) AND #tempJogBackward)) // double negative -> positive direction
	                      THEN
	                        // Positive direction
	                        IF (#stat5D6D) THEN
	                          #tempLimitACJCS := #tempJointUpperLimit[#tempAffectedAxis];
	                        END_IF;
	                        IF (#tempAxisSWLimitActive[#tempAffectedAxis]) THEN
	                          #tempLimitACMCS := #tempAxisSWLimitMaxPos[#tempAffectedAxis];
	                        END_IF;
	                      ELSE
	                        // Negative direction
	                        IF (#stat5D6D) THEN
	                          #tempLimitACJCS := #tempJointLowerLimit[#tempAffectedAxis];
	                        END_IF;
	                        IF (#tempAxisSWLimitActive[#tempAffectedAxis]) THEN
	                          #tempLimitACMCS := #tempAxisSWLimitMinPos[#tempAffectedAxis];
	                        END_IF;
	                      END_IF;
	                      
	                      IF (#stat5D6D) THEN
	                        #tempDistToLimitACJCS := ABS((#tempLimitACJCS - #tempJointPosition[#tempAffectedAxis]) / #tempFactor);
	                      END_IF;
	                      
	                      IF (#tempAxisSWLimitActive[#tempAffectedAxis]) THEN
	                        #tempDistToLimitACMCS := ABS((#tempLimitACMCS - #tempAxisPosition[#tempAffectedAxis]) / #tempFactor);
	                      ELSE
	                        #tempDistToLimitACMCS := #MAX_DISTANCE;
	                      END_IF;
	                      
	                      #tempDistToLimitACMin := MIN(IN1 := #tempDistToLimitACMin, IN2 := #tempDistToLimitACJCS, IN3 := #tempDistToLimitACMCS);
	                    END_FOR;
	                    
	                    // Reduce to distance limit (e.g. relative)
	                    #tempDistToLimit := MIN(IN1 := #tempDistToLimitACMin, IN2 := #tempDistToLimit);
	                    
	                    // Invert solution for negative direction
	                    IF (#tempJogBackward) THEN
	                      #tempDistToLimit *= -1.0;
	                    END_IF;
	                    
	                    #instMC_MoveDirectRelative.Distance[#jogDirection] := #tempDistToLimit;
	                  ELSE
	                    #instMC_MoveDirectRelative.Distance[#jogDirection] := 0.0;
	                  END_IF;
	                  
	                ELSE
	                  // set MC_MoveLinearRelative parameter
	                  #instMC_MoveLinearRelative.CoordSystem := #coordSystem;
	                  #instMC_MoveLinearRelative.Velocity := #dynamics.path.velocity;
	                  #instMC_MoveLinearRelative.Acceleration := #dynamics.path.acceleration;
	                  #instMC_MoveLinearRelative.Deceleration := #dynamics.path.deceleration;
	                  #instMC_MoveLinearRelative.Jerk := #dynamics.path.jerk;
	                  
	                  // initialize jog distance - clear old values
	                  FOR #tempCounter := 1 TO 6 DO
	                    #instMC_MoveLinearRelative.Distance[#tempCounter] := 0.0;
	                  END_FOR;
	                  
	                  // set distance at command
	                  #instMC_MoveLinearRelative.Distance[#jogDirection] := #tempJogDistance;
	                  
